LIN {X 0,Y 488.936,Z 692.562,A -85,B 0,C 180,E1 -6380.904,E2 -6380.904} C_VEL
LIN {X 0,Y 488.778,Z 691.698,A -85,B 0,C 180,E1 -6381.057,E2 -6381.057} C_VEL
LIN {X 0,Y 488.78,Z 691.596,A -85,B 0,C 180,E1 -6383.396,E2 -6383.396} C_VEL
LIN {X 0,Y 488.666,Z 691.611,A -85,B 0,C 180,E1 -6385.878,E2 -6385.878} C_VEL
LIN {X 0,Y 488.944,Z 691.579,A -85,B 0,C 180,E1 -6387.53,E2 -6387.53} C_VEL
LIN {X 0,Y 488.944,Z 691.581,A -85,B 0,C 180,E1 -6390.001,E2 -6390.001} C_VEL
LIN {X 0,Y 488.943,Z 691.584,A -85,B 0,C 180,E1 -6392.473,E2 -6392.473} C_VEL
LIN {X 0,Y 488.815,Z 691.594,A -85,B 0,C 180,E1 -6395.777,E2 -6395.777} C_VEL
LIN {X 0,Y 488.758,Z 691.602,A -85,B 0,C 180,E1 -6398.269,E2 -6398.269} C_VEL
LIN {X 0,Y 488.778,Z 691.595,A -85,B 0,C 180,E1 -6401.614,E2 -6401.614} C_VEL
LIN {X 0,Y 488.759,Z 691.601,A -85,B 0,C 180,E1 -6405.002,E2 -6405.002} C_VEL
LIN {X 0,Y 488.72,Z 691.607,A -85,B 0,C 180,E1 -6408.445,E2 -6408.445} C_VEL
LIN {X 0,Y 488.708,Z 691.61,A -85,B 0,C 180,E1 -6411.072,E2 -6411.072} C_VEL
LIN {X 0,Y 488.668,Z 691.61,A -85,B 0,C 180,E1 -6413.748,E2 -6413.748} C_VEL
LIN {X 0,Y 488.673,Z 691.604,A -85,B 0,C 180,E1 -6416.478,E2 -6416.478} C_VEL
LIN {X 0,Y 488.664,Z 691.617,A -85,B 0,C 180,E1 -6419.275,E2 -6419.275} C_VEL
LIN {X 0,Y 488.684,Z 691.605,A -85,B 0,C 180,E1 -6422.15,E2 -6422.15} C_VEL
LIN {X 0,Y 488.7,Z 691.599,A -85,B 0,C 180,E1 -6425.118,E2 -6425.118} C_VEL
LIN {X 0,Y 488.649,Z 691.611,A -85,B 0,C 180,E1 -6428.204,E2 -6428.204} C_VEL
LIN {X 0,Y 488.648,Z 691.62,A -85,B 0,C 180,E1 -6431.423,E2 -6431.423} C_VEL
LIN {X 0,Y 488.702,Z 691.606,A -85,B 0,C 180,E1 -6434.804,E2 -6434.804} C_VEL
LIN {X 0,Y 488.654,Z 691.617,A -85,B 0,C 180,E1 -6437.47,E2 -6437.47} C_VEL
LIN {X 0,Y 488.671,Z 691.61,A -85,B 0,C 180,E1 -6440.742,E2 -6440.742} C_VEL
LIN {X 0,Y 488.637,Z 691.621,A -85,B 0,C 180,E1 -6443.864,E2 -6443.864} C_VEL
LIN {X 0,Y 488.684,Z 691.61,A -85,B 0,C 180,E1 -6446.873,E2 -6446.873} C_VEL
LIN {X 0,Y 488.67,Z 691.617,A -85,B 0,C 180,E1 -6449.777,E2 -6449.777} C_VEL
LIN {X 0,Y 488.735,Z 691.812,A -85,B 0,C 180,E1 -6451.191,E2 -6451.191} C_VEL
LIN {X 0,Y 488.91,Z 692.685,A -85,B 0,C 180,E1 -6451.311,E2 -6451.311} C_VEL
LIN {X 0,Y 491.517,Z 700.39,A -85,B 0,C 180,E1 -6451.531,E2 -6451.531} C_VEL
LIN {X 0,Y 491.069,Z 767.576,A -85,B 0,C 180,E1 -6452.576,E2 -6452.576} C_VEL
LIN {X 0,Y 490.938,Z 778.889,A -85,B 0,C 180,E1 -6452.88,E2 -6452.88} C_VEL
LIN {X 0,Y 490.731,Z 789.801,A -85,B 0,C 180,E1 -6453.299,E2 -6453.299} C_VEL
LIN {X 0,Y 490.544,Z 798.848,A -85,B 0,C 180,E1 -6453.746,E2 -6453.746} C_VEL
LIN {X 0,Y 490.248,Z 807.955,A -85,B 0,C 180,E1 -6454.3,E2 -6454.3} C_VEL
LIN {X 0,Y 489.93,Z 818.39,A -85,B 0,C 180,E1 -6455.097,E2 -6455.097} C_VEL
LIN {X 0,Y 489.601,Z 826.602,A -85,B 0,C 180,E1 -6455.851,E2 -6455.851} C_VEL
LIN {X 0,Y 489.333,Z 835.233,A -85,B 0,C 180,E1 -6456.811,E2 -6456.811} C_VEL
LIN {X 0,Y 489.045,Z 842.903,A -85,B 0,C 180,E1 -6457.837,E2 -6457.837} C_VEL
LIN {X 0,Y 488.795,Z 848.474,A -85,B 0,C 180,E1 -6458.712,E2 -6458.712} C_VEL
LIN {X 0,Y 488.607,Z 854.255,A -85,B 0,C 180,E1 -6459.805,E2 -6459.805} C_VEL
LIN {X 0,Y 488.459,Z 859.764,A -85,B 0,C 180,E1 -6461.111,E2 -6461.111} C_VEL
LIN {X 0,Y 488.295,Z 864.002,A -85,B 0,C 180,E1 -6462.407,E2 -6462.407} C_VEL
LIN {X 0,Y 488.208,Z 866.278,A -85,B 0,C 180,E1 -6463.267,E2 -6463.267} C_VEL
LIN {X 0,Y 488.154,Z 868.86,A -85,B 0,C 180,E1 -6464.713,E2 -6464.713} C_VEL
LIN {X 0,Y 488.118,Z 870.091,A -85,B 0,C 180,E1 -6465.832,E2 -6465.832} C_VEL
LIN {X 0,Y 488.143,Z 870.488,A -85,B 0,C 180,E1 -6466.682,E2 -6466.682} C_VEL
LIN {X 0,Y 488.181,Z 870.191,A -85,B 0,C 180,E1 -6468.227,E2 -6468.227} C_VEL
LIN {X 0,Y 488.214,Z 869.199,A -85,B 0,C 180,E1 -6469.214,E2 -6469.214} C_VEL
LIN {X 0,Y 488.29,Z 866.395,A -85,B 0,C 180,E1 -6470.89,E2 -6470.89} C_VEL
LIN {X 0,Y 488.444,Z 863.069,A -85,B 0,C 180,E1 -6472.143,E2 -6472.143} C_VEL
LIN {X 0,Y 488.58,Z 858.666,A -85,B 0,C 180,E1 -6473.392,E2 -6473.392} C_VEL
LIN {X 0,Y 488.736,Z 853.034,A -85,B 0,C 180,E1 -6474.637,E2 -6474.637} C_VEL
LIN {X 0,Y 488.912,Z 847.33,A -85,B 0,C 180,E1 -6475.672,E2 -6475.672} C_VEL
LIN {X 0,Y 489.218,Z 840.419,A -85,B 0,C 180,E1 -6476.706,E2 -6476.706} C_VEL
LIN {X 0,Y 489.54,Z 832.033,A -85,B 0,C 180,E1 -6477.737,E2 -6477.737} C_VEL
LIN {X 0,Y 489.821,Z 824.016,A -85,B 0,C 180,E1 -6478.561,E2 -6478.561} C_VEL
LIN {X 0,Y 490.161,Z 814.265,A -85,B 0,C 180,E1 -6479.384,E2 -6479.384} C_VEL
LIN {X 0,Y 490.428,Z 805.41,A -85,B 0,C 180,E1 -6480,E2 -6480} C_VEL
LIN {X 0,Y 490.655,Z 795.361,A -85,B 0,C 180,E1 -6480.564,E2 -6480.564} C_VEL
LIN {X 0,Y 490.911,Z 784.684,A -85,B 0,C 180,E1 -6481.025,E2 -6481.025} C_VEL
LIN {X 0,Y 491.017,Z 774.27,A -85,B 0,C 180,E1 -6481.358,E2 -6481.358} C_VEL
LIN {X 0,Y 491.113,Z 762.086,A -85,B 0,C 180,E1 -6481.614,E2 -6481.614} C_VEL
LIN {X 0,Y 491.441,Z 699.545,A -85,B 0,C 180,E1 -6482.577,E2 -6482.577} C_VEL
LIN {X 0,Y 489.035,Z 692.377,A -85,B 0,C 180,E1 -6482.806,E2 -6482.806} C_VEL
LIN {X 0,Y 488.882,Z 691.641,A -85,B 0,C 180,E1 -6482.987,E2 -6482.987} C_VEL
LIN {X 0,Y 488.844,Z 691.595,A -85,B 0,C 180,E1 -6485.776,E2 -6485.776} C_VEL
LIN {X 0,Y 488.792,Z 691.601,A -85,B 0,C 180,E1 -6488.267,E2 -6488.267} C_VEL
LIN {X 0,Y 488.812,Z 691.595,A -85,B 0,C 180,E1 -6491.612,E2 -6491.612} C_VEL
LIN {X 0,Y 488.769,Z 691.6,A -85,B 0,C 180,E1 -6495,E2 -6495} C_VEL
LIN {X 0,Y 488.754,Z 691.607,A -85,B 0,C 180,E1 -6498.442,E2 -6498.442} C_VEL
LIN {X 0,Y 488.714,Z 691.607,A -85,B 0,C 180,E1 -6501.07,E2 -6501.07} C_VEL
LIN {X 0,Y 488.69,Z 691.607,A -85,B 0,C 180,E1 -6503.746,E2 -6503.746} C_VEL
LIN {X 0,Y 488.732,Z 691.609,A -85,B 0,C 180,E1 -6506.928,E2 -6506.928} C_VEL
LIN {X 0,Y 488.731,Z 691.604,A -85,B 0,C 180,E1 -6510.219,E2 -6510.219} C_VEL
LIN {X 0,Y 488.735,Z 691.604,A -85,B 0,C 180,E1 -6513.483,E2 -6513.483} C_VEL
LIN {X 0,Y 488.688,Z 691.609,A -85,B 0,C 180,E1 -6516.354,E2 -6516.354} C_VEL
LIN {X 0,Y 488.707,Z 691.612,A -85,B 0,C 180,E1 -6519.254,E2 -6519.254} C_VEL
LIN {X 0,Y 488.713,Z 691.609,A -85,B 0,C 180,E1 -6521.599,E2 -6521.599} C_VEL
LIN {X 0,Y 488.708,Z 691.608,A -85,B 0,C 180,E1 -6524.802,E2 -6524.802} C_VEL
LIN {X 0,Y 488.698,Z 691.614,A -85,B 0,C 180,E1 -6527.474,E2 -6527.474} C_VEL
LIN {X 0,Y 488.739,Z 691.607,A -85,B 0,C 180,E1 -6529.676,E2 -6529.676} C_VEL
LIN {X 0,Y 488.676,Z 691.61,A -85,B 0,C 180,E1 -6532.84,E2 -6532.84} C_VEL
LIN {X 0,Y 488.729,Z 691.609,A -85,B 0,C 180,E1 -6535.886,E2 -6535.886} C_VEL
LIN {X 0,Y 488.698,Z 691.612,A -85,B 0,C 180,E1 -6538.819,E2 -6538.819} C_VEL
LIN {X 0,Y 488.803,Z 691.843,A -85,B 0,C 180,E1 -6540.068,E2 -6540.068} C_VEL
LIN {X 0,Y 492.608,Z 708.802,A -85,B 0,C 180,E1 -6542.527,E2 -6542.527} C_VEL
LIN {X 0,Y 491.674,Z 731.997,A -85,B 0,C 180,E1 -6545.509,E2 -6545.509} C_VEL
LIN {X 0,Y 490.938,Z 754.807,A -85,B 0,C 180,E1 -6548.401,E2 -6548.401} C_VEL
LIN {X 0,Y 490.099,Z 782.413,A -85,B 0,C 180,E1 -6551.825,E2 -6551.825} C_VEL
LIN {X 0,Y 489.619,Z 797.491,A -85,B 0,C 180,E1 -6553.682,E2 -6553.682} C_VEL
LIN {X 0,Y 490.629,Z 806.708,A -85,B 0,C 180,E1 -6553.883,E2 -6553.883} C_VEL
LIN {X 0,Y 491.648,Z 815.903,A -85,B 0,C 180,E1 -6554.053,E2 -6554.053} C_VEL
LIN {X 0,Y 491.061,Z 909.011,A -85,B 0,C 180,E1 -6555.441,E2 -6555.441} C_VEL
LIN {X 0,Y 490.661,Z 922.838,A -85,B 0,C 180,E1 -6555.826,E2 -6555.826} C_VEL
LIN {X 0,Y 490.322,Z 935.816,A -85,B 0,C 180,E1 -6556.372,E2 -6556.372} C_VEL
LIN {X 0,Y 489.911,Z 948.159,A -85,B 0,C 180,E1 -6557.077,E2 -6557.077} C_VEL
LIN {X 0,Y 489.566,Z 959.167,A -85,B 0,C 180,E1 -6557.879,E2 -6557.879} C_VEL
LIN {X 0,Y 489.119,Z 969.532,A -85,B 0,C 180,E1 -6558.814,E2 -6558.814} C_VEL
LIN {X 0,Y 488.807,Z 978.886,A -85,B 0,C 180,E1 -6559.854,E2 -6559.854} C_VEL
LIN {X 0,Y 488.488,Z 988.009,A -85,B 0,C 180,E1 -6561.102,E2 -6561.102} C_VEL
LIN {X 0,Y 488.265,Z 995.37,A -85,B 0,C 180,E1 -6562.348,E2 -6562.348} C_VEL
LIN {X 0,Y 488.141,Z 1001.708,A -85,B 0,C 180,E1 -6563.703,E2 -6563.703} C_VEL
LIN {X 0,Y 488.037,Z 1006.546,A -85,B 0,C 180,E1 -6565.042,E2 -6565.042} C_VEL
LIN {X 0,Y 488.031,Z 1008.908,A -85,B 0,C 180,E1 -6565.87,E2 -6565.87} C_VEL
LIN {X 0,Y 488.029,Z 1010.823,A -85,B 0,C 180,E1 -6566.697,E2 -6566.697} C_VEL
LIN {X 0,Y 487.977,Z 1012.255,A -85,B 0,C 180,E1 -6567.522,E2 -6567.522} C_VEL
LIN {X 0,Y 487.951,Z 1013.276,A -85,B 0,C 180,E1 -6568.348,E2 -6568.348} C_VEL
LIN {X 0,Y 487.913,Z 1013.895,A -85,B 0,C 180,E1 -6569.173,E2 -6569.173} C_VEL
LIN {X 0,Y 487.905,Z 1014.113,A -85,B 0,C 180,E1 -6569.999,E2 -6569.999} C_VEL
LIN {X 0,Y 487.914,Z 1013.89,A -85,B 0,C 180,E1 -6570.824,E2 -6570.824} C_VEL
LIN {X 0,Y 487.952,Z 1013.268,A -85,B 0,C 180,E1 -6571.649,E2 -6571.649} C_VEL
LIN {X 0,Y 487.978,Z 1012.243,A -85,B 0,C 180,E1 -6572.475,E2 -6572.475} C_VEL
LIN {X 0,Y 488.028,Z 1010.805,A -85,B 0,C 180,E1 -6573.301,E2 -6573.301} C_VEL
LIN {X 0,Y 488.02,Z 1007.773,A -85,B 0,C 180,E1 -6574.542,E2 -6574.542} C_VEL
LIN {X 0,Y 488.139,Z 1003.69,A -85,B 0,C 180,E1 -6575.783,E2 -6575.783} C_VEL
LIN {X 0,Y 488.188,Z 997.396,A -85,B 0,C 180,E1 -6577.235,E2 -6577.235} C_VEL
LIN {X 0,Y 488.418,Z 990.553,A -85,B 0,C 180,E1 -6578.48,E2 -6578.48} C_VEL
LIN {X 0,Y 488.674,Z 982.07,A -85,B 0,C 180,E1 -6579.728,E2 -6579.728} C_VEL
LIN {X 0,Y 488.946,Z 973.387,A -85,B 0,C 180,E1 -6580.768,E2 -6580.768} C_VEL
LIN {X 0,Y 489.38,Z 962.702,A -85,B 0,C 180,E1 -6581.807,E2 -6581.807} C_VEL
LIN {X 0,Y 489.823,Z 951.136,A -85,B 0,C 180,E1 -6582.711,E2 -6582.711} C_VEL
LIN {X 0,Y 490.176,Z 938.635,A -85,B 0,C 180,E1 -6583.472,E2 -6583.472} C_VEL
LIN {X 0,Y 490.612,Z 926.141,A -85,B 0,C 180,E1 -6584.04,E2 -6584.04} C_VEL
LIN {X 0,Y 490.952,Z 913.323,A -85,B 0,C 180,E1 -6584.454,E2 -6584.454} C_VEL
LIN {X 0,Y 491.139,Z 898.092,A -85,B 0,C 180,E1 -6584.739,E2 -6584.739} C_VEL
LIN {X 0,Y 491.615,Z 814.3,A -85,B 0,C 180,E1 -6585.966,E2 -6585.966} C_VEL
LIN {X 0,Y 489.61,Z 797.388,A -85,B 0,C 180,E1 -6586.296,E2 -6586.296} C_VEL
LIN {X 0,Y 490.203,Z 775.247,A -85,B 0,C 180,E1 -6588.998,E2 -6588.998} C_VEL
LIN {X 0,Y 490.964,Z 750.475,A -85,B 0,C 180,E1 -6592.07,E2 -6592.07} C_VEL
LIN {X 0,Y 491.789,Z 726.02,A -85,B 0,C 180,E1 -6595.158,E2 -6595.158} C_VEL
LIN {X 0,Y 492.452,Z 708.982,A -85,B 0,C 180,E1 -6597.346,E2 -6597.346} C_VEL
LIN {X 0,Y 490.614,Z 699.96,A -85,B 0,C 180,E1 -6598.62,E2 -6598.62} C_VEL
LIN {X 0,Y 488.756,Z 691.718,A -85,B 0,C 180,E1 -6599.859,E2 -6599.859} C_VEL
LIN {X 0,Y 488.733,Z 691.605,A -85,B 0,C 180,E1 -6603.121,E2 -6603.121} C_VEL
LIN {X 0,Y 488.671,Z 691.616,A -85,B 0,C 180,E1 -6606.131,E2 -6606.131} C_VEL
LIN {X 0,Y 488.694,Z 691.609,A -85,B 0,C 180,E1 -6609.253,E2 -6609.253} C_VEL
LIN {X 0,Y 488.699,Z 691.607,A -85,B 0,C 180,E1 -6611.599,E2 -6611.599} C_VEL
LIN {X 0,Y 488.704,Z 691.612,A -85,B 0,C 180,E1 -6614.8,E2 -6614.8} C_VEL
LIN {X 0,Y 488.688,Z 691.609,A -85,B 0,C 180,E1 -6617.474,E2 -6617.474} C_VEL
LIN {X 0,Y 488.724,Z 691.598,A -85,B 0,C 180,E1 -6619.676,E2 -6619.676} C_VEL
LIN {X 0,Y 488.673,Z 691.616,A -85,B 0,C 180,E1 -6622.84,E2 -6622.84} C_VEL
LIN {X 0,Y 488.725,Z 691.602,A -85,B 0,C 180,E1 -6625.887,E2 -6625.887} C_VEL
LIN {X 0,Y 488.685,Z 691.61,A -85,B 0,C 180,E1 -6628.82,E2 -6628.82} C_VEL
LIN {X 0,Y 488.736,Z 691.604,A -85,B 0,C 180,E1 -6631.671,E2 -6631.671} C_VEL
LIN {X 0,Y 488.74,Z 691.6,A -85,B 0,C 180,E1 -6634.444,E2 -6634.444} C_VEL
LIN {X 0,Y 488.71,Z 691.608,A -85,B 0,C 180,E1 -6637.153,E2 -6637.153} C_VEL
LIN {X 0,Y 488.713,Z 691.611,A -85,B 0,C 180,E1 -6639.81,E2 -6639.81} C_VEL
LIN {X 0,Y 488.722,Z 691.6,A -85,B 0,C 180,E1 -6642.423,E2 -6642.423} C_VEL
LIN {X 0,Y 488.75,Z 691.6,A -85,B 0,C 180,E1 -6644.999,E2 -6644.999} C_VEL
LIN {X 0,Y 488.793,Z 691.597,A -85,B 0,C 180,E1 -6648.387,E2 -6648.387} C_VEL
LIN {X 0,Y 488.805,Z 691.592,A -85,B 0,C 180,E1 -6651.734,E2 -6651.734} C_VEL
LIN {X 0,Y 488.836,Z 691.594,A -85,B 0,C 180,E1 -6654.224,E2 -6654.224} C_VEL
LIN {X 0,Y 488.948,Z 691.574,A -85,B 0,C 180,E1 -6657.529,E2 -6657.529} C_VEL
LIN {X 0,Y 488.943,Z 691.577,A -85,B 0,C 180,E1 -6660.824,E2 -6660.824} C_VEL
LIN {X 0,Y 488.948,Z 691.583,A -85,B 0,C 180,E1 -6662.472,E2 -6662.472} C_VEL
LIN {X 0,Y 488.836,Z 691.588,A -85,B 0,C 180,E1 -6665.776,E2 -6665.776} C_VEL
LIN {X 0,Y 488.806,Z 691.595,A -85,B 0,C 180,E1 -6668.267,E2 -6668.267} C_VEL
LIN {X 0,Y 488.796,Z 691.593,A -85,B 0,C 180,E1 -6671.613,E2 -6671.613} C_VEL
LIN {X 0,Y 488.75,Z 691.605,A -85,B 0,C 180,E1 -6675.001,E2 -6675.001} C_VEL
LIN {X 0,Y 488.735,Z 691.603,A -85,B 0,C 180,E1 -6678.443,E2 -6678.443} C_VEL
LIN {X 0,Y 488.695,Z 691.615,A -85,B 0,C 180,E1 -6681.072,E2 -6681.072} C_VEL
LIN {X 0,Y 488.661,Z 691.608,A -85,B 0,C 180,E1 -6683.747,E2 -6683.747} C_VEL
LIN {X 0,Y 488.737,Z 691.606,A -85,B 0,C 180,E1 -6686.934,E2 -6686.934} C_VEL
LIN {X 0,Y 488.712,Z 691.605,A -85,B 0,C 180,E1 -6689.271,E2 -6689.271} C_VEL
LIN {X 0,Y 488.694,Z 691.604,A -85,B 0,C 180,E1 -6692.148,E2 -6692.148} C_VEL
LIN {X 0,Y 488.713,Z 691.608,A -85,B 0,C 180,E1 -6695.116,E2 -6695.116} C_VEL
LIN {X 0,Y 488.672,Z 691.61,A -85,B 0,C 180,E1 -6698.201,E2 -6698.201} C_VEL
LIN {X 0,Y 488.71,Z 691.607,A -85,B 0,C 180,E1 -6700.346,E2 -6700.346} C_VEL
LIN {X 0,Y 488.677,Z 691.614,A -85,B 0,C 180,E1 -6703.656,E2 -6703.656} C_VEL
LIN {X 0,Y 488.671,Z 691.609,A -85,B 0,C 180,E1 -6706.346,E2 -6706.346} C_VEL
LIN {X 0,Y 488.772,Z 691.798,A -85,B 0,C 180,E1 -6709.048,E2 -6709.048} C_VEL
LIN {X 0,Y 489.014,Z 692.905,A -85,B 0,C 180,E1 -6709.184,E2 -6709.184} C_VEL
LIN {X 0,Y 491.909,Z 700.992,A -85,B 0,C 180,E1 -6709.415,E2 -6709.415} C_VEL
LIN {X 0,Y 491.437,Z 772.238,A -85,B 0,C 180,E1 -6710.494,E2 -6710.494} C_VEL
LIN {X 0,Y 491.368,Z 785.777,A -85,B 0,C 180,E1 -6710.878,E2 -6710.878} C_VEL
LIN {X 0,Y 491.208,Z 797.787,A -85,B 0,C 180,E1 -6711.381,E2 -6711.381} C_VEL
LIN {X 0,Y 490.972,Z 807.684,A -85,B 0,C 180,E1 -6711.928,E2 -6711.928} C_VEL
LIN {X 0,Y 490.236,Z 812.918,A -85,B 0,C 180,E1 -6712.238,E2 -6712.238} C_VEL
LIN {X 0,Y 487.217,Z 821.277,A -85,B 0,C 180,E1 -6712.758,E2 -6712.758} C_VEL
LIN {X 0,Y 484.13,Z 829.158,A -85,B 0,C 180,E1 -6713.365,E2 -6713.365} C_VEL
LIN {X 0,Y 483.294,Z 833.637,A -85,B 0,C 180,E1 -6713.808,E2 -6713.808} C_VEL
LIN {X 0,Y 482.865,Z 842.864,A -85,B 0,C 180,E1 -6714.908,E2 -6714.908} C_VEL
LIN {X 0,Y 482.444,Z 851.205,A -85,B 0,C 180,E1 -6716.135,E2 -6716.135} C_VEL
LIN {X 0,Y 482.214,Z 857.921,A -85,B 0,C 180,E1 -6717.369,E2 -6717.369} C_VEL
LIN {X 0,Y 481.878,Z 864.127,A -85,B 0,C 180,E1 -6718.82,E2 -6718.82} C_VEL
LIN {X 0,Y 481.67,Z 868.785,A -85,B 0,C 180,E1 -6720.26,E2 -6720.26} C_VEL
LIN {X 0,Y 481.557,Z 871.112,A -85,B 0,C 180,E1 -6721.211,E2 -6721.211} C_VEL
LIN {X 0,Y 481.484,Z 872.871,A -85,B 0,C 180,E1 -6722.156,E2 -6722.156} C_VEL
LIN {X 0,Y 481.455,Z 874.126,A -85,B 0,C 180,E1 -6723.096,E2 -6723.096} C_VEL
LIN {X 0,Y 481.39,Z 874.851,A -85,B 0,C 180,E1 -6724.026,E2 -6724.026} C_VEL
LIN {X 0,Y 481.378,Z 875.127,A -85,B 0,C 180,E1 -6724.953,E2 -6724.953} C_VEL
LIN {X 0,Y 481.359,Z 874.918,A -85,B 0,C 180,E1 -6725.872,E2 -6725.872} C_VEL
LIN {X 0,Y 481.396,Z 874.137,A -85,B 0,C 180,E1 -6726.891,E2 -6726.891} C_VEL
LIN {X 0,Y 481.44,Z 873.13,A -85,B 0,C 180,E1 -6727.696,E2 -6727.696} C_VEL
LIN {X 0,Y 481.603,Z 870.535,A -85,B 0,C 180,E1 -6729.06,E2 -6729.06} C_VEL
LIN {X 0,Y 481.73,Z 866.893,A -85,B 0,C 180,E1 -6730.396,E2 -6730.396} C_VEL
LIN {X 0,Y 481.967,Z 861.718,A -85,B 0,C 180,E1 -6731.804,E2 -6731.804} C_VEL
LIN {X 0,Y 482.226,Z 854.725,A -85,B 0,C 180,E1 -6733.273,E2 -6733.273} C_VEL
LIN {X 0,Y 482.587,Z 847.687,A -85,B 0,C 180,E1 -6734.441,E2 -6734.441} C_VEL
LIN {X 0,Y 482.958,Z 838.437,A -85,B 0,C 180,E1 -6735.679,E2 -6735.679} C_VEL
LIN {X 0,Y 483.355,Z 829.161,A -85,B 0,C 180,E1 -6736.684,E2 -6736.684} C_VEL
LIN {X 0,Y 483.733,Z 818.409,A -85,B 0,C 180,E1 -6737.627,E2 -6737.627} C_VEL
LIN {X 0,Y 484.076,Z 807.541,A -85,B 0,C 180,E1 -6738.38,E2 -6738.38} C_VEL
LIN {X 0,Y 484.32,Z 795.637,A -85,B 0,C 180,E1 -6739.022,E2 -6739.022} C_VEL
LIN {X 0,Y 484.505,Z 782.745,A -85,B 0,C 180,E1 -6739.528,E2 -6739.528} C_VEL
LIN {X 0,Y 484.6,Z 770.059,A -85,B 0,C 180,E1 -6739.847,E2 -6739.847} C_VEL
LIN {X 0,Y 484.959,Z 702.07,A -85,B 0,C 180,E1 -6740.876,E2 -6740.876} C_VEL
LIN {X 0,Y 481.891,Z 693.353,A -85,B 0,C 180,E1 -6741.148,E2 -6741.148} C_VEL
LIN {X 0,Y 481.733,Z 692.534,A -85,B 0,C 180,E1 -6741.327,E2 -6741.327} C_VEL
LIN {X 0,Y 481.777,Z 692.474,A -85,B 0,C 180,E1 -6744.14,E2 -6744.14} C_VEL
LIN {X 0,Y 481.909,Z 692.456,A -85,B 0,C 180,E1 -6747.494,E2 -6747.494} C_VEL
LIN {X 0,Y 481.913,Z 692.457,A -85,B 0,C 180,E1 -6750.001,E2 -6750.001} C_VEL
LIN {X 0,Y 481.908,Z 692.46,A -85,B 0,C 180,E1 -6752.509,E2 -6752.509} C_VEL
LIN {X 0,Y 481.777,Z 692.471,A -85,B 0,C 180,E1 -6755.862,E2 -6755.862} C_VEL
LIN {X 0,Y 481.716,Z 692.481,A -85,B 0,C 180,E1 -6758.39,E2 -6758.39} C_VEL
LIN {X 0,Y 481.729,Z 692.473,A -85,B 0,C 180,E1 -6761.787,E2 -6761.787} C_VEL
LIN {X 0,Y 481.743,Z 692.472,A -85,B 0,C 180,E1 -6765.225,E2 -6765.225} C_VEL
LIN {X 0,Y 481.663,Z 692.487,A -85,B 0,C 180,E1 -6768.725,E2 -6768.725} C_VEL
LIN {X 0,Y 481.647,Z 692.486,A -85,B 0,C 180,E1 -6771.396,E2 -6771.396} C_VEL
LIN {X 0,Y 481.647,Z 692.484,A -85,B 0,C 180,E1 -6774.116,E2 -6774.116} C_VEL
LIN {X 0,Y 481.647,Z 692.483,A -85,B 0,C 180,E1 -6777.115,E2 -6777.115} C_VEL
LIN {X 0,Y 481.605,Z 692.491,A -85,B 0,C 180,E1 -6779.747,E2 -6779.747} C_VEL
LIN {X 0,Y 481.639,Z 692.484,A -85,B 0,C 180,E1 -6782.678,E2 -6782.678} C_VEL
LIN {X 0,Y 481.644,Z 692.478,A -85,B 0,C 180,E1 -6785.2,E2 -6785.2} C_VEL
LIN {X 0,Y 481.626,Z 692.487,A -85,B 0,C 180,E1 -6788.002,E2 -6788.002} C_VEL
LIN {X 0,Y 481.609,Z 692.491,A -85,B 0,C 180,E1 -6791.048,E2 -6791.048} C_VEL
LIN {X 0,Y 481.638,Z 692.485,A -85,B 0,C 180,E1 -6794.461,E2 -6794.461} C_VEL
LIN {X 0,Y 481.618,Z 692.488,A -85,B 0,C 180,E1 -6796.856,E2 -6796.856} C_VEL
LIN {X 0,Y 481.633,Z 692.492,A -85,B 0,C 180,E1 -6800.055,E2 -6800.055} C_VEL
LIN {X 0,Y 481.602,Z 692.492,A -85,B 0,C 180,E1 -6803.251,E2 -6803.251} C_VEL
LIN {X 0,Y 481.678,Z 692.487,A -85,B 0,C 180,E1 -6806.327,E2 -6806.327} C_VEL
LIN {X 0,Y 481.617,Z 692.494,A -85,B 0,C 180,E1 -6809.426,E2 -6809.426} C_VEL
LIN {X 0,Y 481.68,Z 692.657,A -85,B 0,C 180,E1 -6810.951,E2 -6810.951} C_VEL
LIN {X 0,Y 481.895,Z 693.673,A -85,B 0,C 180,E1 -6811.09,E2 -6811.09} C_VEL
LIN {X 0,Y 484.721,Z 701.805,A -85,B 0,C 180,E1 -6811.327,E2 -6811.327} C_VEL
LIN {X 0,Y 484.189,Z 768.388,A -85,B 0,C 180,E1 -6812.382,E2 -6812.382} C_VEL
LIN {X 0,Y 484.073,Z 779.919,A -85,B 0,C 180,E1 -6812.697,E2 -6812.697} C_VEL
LIN {X 0,Y 483.85,Z 790.799,A -85,B 0,C 180,E1 -6813.121,E2 -6813.121} C_VEL
LIN {X 0,Y 483.662,Z 799.838,A -85,B 0,C 180,E1 -6813.576,E2 -6813.576} C_VEL
LIN {X 0,Y 483.368,Z 808.945,A -85,B 0,C 180,E1 -6814.139,E2 -6814.139} C_VEL
LIN {X 0,Y 483.062,Z 818.474,A -85,B 0,C 180,E1 -6814.866,E2 -6814.866} C_VEL
LIN {X 0,Y 482.688,Z 827.593,A -85,B 0,C 180,E1 -6815.712,E2 -6815.712} C_VEL
LIN {X 0,Y 482.43,Z 835.608,A -85,B 0,C 180,E1 -6816.605,E2 -6816.605} C_VEL
LIN {X 0,Y 482.175,Z 842.456,A -85,B 0,C 180,E1 -6817.504,E2 -6817.504} C_VEL
LIN {X 0,Y 481.819,Z 849.481,A -85,B 0,C 180,E1 -6818.613,E2 -6818.613} C_VEL
LIN {X 0,Y 481.657,Z 854.26,A -85,B 0,C 180,E1 -6819.501,E2 -6819.501} C_VEL
LIN {X 0,Y 481.498,Z 860.012,A -85,B 0,C 180,E1 -6820.827,E2 -6820.827} C_VEL
LIN {X 0,Y 481.32,Z 864.44,A -85,B 0,C 180,E1 -6822.143,E2 -6822.143} C_VEL
LIN {X 0,Y 481.205,Z 866.797,A -85,B 0,C 180,E1 -6823.016,E2 -6823.016} C_VEL
LIN {X 0,Y 481.141,Z 869.948,A -85,B 0,C 180,E1 -6824.756,E2 -6824.756} C_VEL
LIN {X 0,Y 481.1,Z 870.954,A -85,B 0,C 180,E1 -6825.621,E2 -6825.621} C_VEL
LIN {X 0,Y 481.122,Z 871.467,A -85,B 0,C 180,E1 -6826.484,E2 -6826.484} C_VEL
LIN {X 0,Y 481.179,Z 871.245,A -85,B 0,C 180,E1 -6828.201,E2 -6828.201} C_VEL
LIN {X 0,Y 481.224,Z 869.341,A -85,B 0,C 180,E1 -6829.906,E2 -6829.906} C_VEL
LIN {X 0,Y 481.301,Z 866.839,A -85,B 0,C 180,E1 -6831.18,E2 -6831.18} C_VEL
LIN {X 0,Y 481.489,Z 863.306,A -85,B 0,C 180,E1 -6832.451,E2 -6832.451} C_VEL
LIN {X 0,Y 481.652,Z 858.673,A -85,B 0,C 180,E1 -6833.717,E2 -6833.717} C_VEL
LIN {X 0,Y 481.779,Z 853.92,A -85,B 0,C 180,E1 -6834.769,E2 -6834.769} C_VEL
LIN {X 0,Y 481.98,Z 848.169,A -85,B 0,C 180,E1 -6835.819,E2 -6835.819} C_VEL
LIN {X 0,Y 482.311,Z 841.203,A -85,B 0,C 180,E1 -6836.867,E2 -6836.867} C_VEL
LIN {X 0,Y 482.642,Z 832.757,A -85,B 0,C 180,E1 -6837.914,E2 -6837.914} C_VEL
LIN {X 0,Y 482.951,Z 824.664,A -85,B 0,C 180,E1 -6838.749,E2 -6838.749} C_VEL
LIN {X 0,Y 483.236,Z 816.234,A -85,B 0,C 180,E1 -6839.479,E2 -6839.479} C_VEL
LIN {X 0,Y 483.532,Z 807.575,A -85,B 0,C 180,E1 -6840.104,E2 -6840.104} C_VEL
LIN {X 0,Y 483.785,Z 796.73,A -85,B 0,C 180,E1 -6840.728,E2 -6840.728} C_VEL
LIN {X 0,Y 484.018,Z 786.174,A -85,B 0,C 180,E1 -6841.196,E2 -6841.196} C_VEL
LIN {X 0,Y 484.139,Z 775.934,A -85,B 0,C 180,E1 -6841.534,E2 -6841.534} C_VEL
LIN {X 0,Y 484.266,Z 762.405,A -85,B 0,C 180,E1 -6841.819,E2 -6841.819} C_VEL
LIN {X 0,Y 484.709,Z 701.263,A -85,B 0,C 180,E1 -6842.78,E2 -6842.78} C_VEL
LIN {X 0,Y 482.024,Z 693.475,A -85,B 0,C 180,E1 -6843.02,E2 -6843.02} C_VEL
LIN {X 0,Y 481.805,Z 692.564,A -85,B 0,C 180,E1 -6843.183,E2 -6843.183} C_VEL
LIN {X 0,Y 481.803,Z 692.473,A -85,B 0,C 180,E1 -6845.86,E2 -6845.86} C_VEL
LIN {X 0,Y 481.746,Z 692.478,A -85,B 0,C 180,E1 -6848.388,E2 -6848.388} C_VEL
LIN {X 0,Y 481.758,Z 692.475,A -85,B 0,C 180,E1 -6851.785,E2 -6851.785} C_VEL
LIN {X 0,Y 481.75,Z 692.473,A -85,B 0,C 180,E1 -6855.224,E2 -6855.224} C_VEL
LIN {X 0,Y 481.715,Z 692.482,A -85,B 0,C 180,E1 -6858.722,E2 -6858.722} C_VEL
LIN {X 0,Y 481.652,Z 692.485,A -85,B 0,C 180,E1 -6861.394,E2 -6861.394} C_VEL
LIN {X 0,Y 481.67,Z 692.484,A -85,B 0,C 180,E1 -6864.113,E2 -6864.113} C_VEL
LIN {X 0,Y 481.701,Z 692.482,A -85,B 0,C 180,E1 -6867.126,E2 -6867.126} C_VEL
LIN {X 0,Y 481.68,Z 692.481,A -85,B 0,C 180,E1 -6869.741,E2 -6869.741} C_VEL
LIN {X 0,Y 481.677,Z 692.486,A -85,B 0,C 180,E1 -6872.674,E2 -6872.674} C_VEL
LIN {X 0,Y 481.642,Z 692.487,A -85,B 0,C 180,E1 -6875.709,E2 -6875.709} C_VEL
LIN {X 0,Y 481.677,Z 692.487,A -85,B 0,C 180,E1 -6878.859,E2 -6878.859} C_VEL
LIN {X 0,Y 481.659,Z 692.485,A -85,B 0,C 180,E1 -6881.912,E2 -6881.912} C_VEL
LIN {X 0,Y 481.661,Z 692.484,A -85,B 0,C 180,E1 -6884.457,E2 -6884.457} C_VEL
LIN {X 0,Y 481.654,Z 692.487,A -85,B 0,C 180,E1 -6887.839,E2 -6887.839} C_VEL
LIN {X 0,Y 481.663,Z 692.483,A -85,B 0,C 180,E1 -6890.654,E2 -6890.654} C_VEL
LIN {X 0,Y 481.628,Z 692.493,A -85,B 0,C 180,E1 -6893.376,E2 -6893.376} C_VEL
LIN {X 0,Y 481.682,Z 692.485,A -85,B 0,C 180,E1 -6896.327,E2 -6896.327} C_VEL
LIN {X 0,Y 481.731,Z 692.662,A -85,B 0,C 180,E1 -6899.809,E2 -6899.809} C_VEL
LIN {X 0,Y 485.708,Z 710.28,A -85,B 0,C 180,E1 -6902.416,E2 -6902.416} C_VEL
LIN {X 0,Y 484.681,Z 734.593,A -85,B 0,C 180,E1 -6905.589,E2 -6905.589} C_VEL
LIN {X 0,Y 483.88,Z 757.058,A -85,B 0,C 180,E1 -6908.475,E2 -6908.475} C_VEL
LIN {X 0,Y 482.979,Z 784.87,A -85,B 0,C 180,E1 -6911.987,E2 -6911.987} C_VEL
LIN {X 0,Y 482.603,Z 796.784,A -85,B 0,C 180,E1 -6913.458,E2 -6913.458} C_VEL
LIN {X 0,Y 484.798,Z 816.369,A -85,B 0,C 180,E1 -6913.843,E2 -6913.843} C_VEL
LIN {X 0,Y 484.168,Z 907.958,A -85,B 0,C 180,E1 -6915.229,E2 -6915.229} C_VEL
LIN {X 0,Y 483.763,Z 921.804,A -85,B 0,C 180,E1 -6915.62,E2 -6915.62} C_VEL
LIN {X 0,Y 483.37,Z 934.791,A -85,B 0,C 180,E1 -6916.172,E2 -6916.172} C_VEL
LIN {X 0,Y 482.917,Z 947.141,A -85,B 0,C 180,E1 -6916.887,E2 -6916.887} C_VEL
LIN {X 0,Y 482.538,Z 958.144,A -85,B 0,C 180,E1 -6917.7,E2 -6917.7} C_VEL
LIN {X 0,Y 482.112,Z 968.519,A -85,B 0,C 180,E1 -6918.649,E2 -6918.649} C_VEL
LIN {X 0,Y 481.728,Z 977.867,A -85,B 0,C 180,E1 -6919.704,E2 -6919.704} C_VEL
LIN {X 0,Y 481.423,Z 986.996,A -85,B 0,C 180,E1 -6920.97,E2 -6920.97} C_VEL
LIN {X 0,Y 481.209,Z 994.362,A -85,B 0,C 180,E1 -6922.235,E2 -6922.235} C_VEL
LIN {X 0,Y 481.077,Z 1001.041,A -85,B 0,C 180,E1 -6923.696,E2 -6923.696} C_VEL
LIN {X 0,Y 480.999,Z 1005.544,A -85,B 0,C 180,E1 -6924.969,E2 -6924.969} C_VEL
LIN {X 0,Y 480.976,Z 1007.903,A -85,B 0,C 180,E1 -6925.809,E2 -6925.809} C_VEL
LIN {X 0,Y 480.984,Z 1009.82,A -85,B 0,C 180,E1 -6926.648,E2 -6926.648} C_VEL
LIN {X 0,Y 480.938,Z 1011.252,A -85,B 0,C 180,E1 -6927.486,E2 -6927.486} C_VEL
LIN {X 0,Y 480.916,Z 1012.273,A -85,B 0,C 180,E1 -6928.324,E2 -6928.324} C_VEL
LIN {X 0,Y 480.883,Z 1012.89,A -85,B 0,C 180,E1 -6929.161,E2 -6929.161} C_VEL
LIN {X 0,Y 480.878,Z 1013.107,A -85,B 0,C 180,E1 -6929.999,E2 -6929.999} C_VEL
LIN {X 0,Y 480.885,Z 1012.882,A -85,B 0,C 180,E1 -6930.836,E2 -6930.836} C_VEL
LIN {X 0,Y 480.919,Z 1012.257,A -85,B 0,C 180,E1 -6931.674,E2 -6931.674} C_VEL
LIN {X 0,Y 480.941,Z 1011.227,A -85,B 0,C 180,E1 -6932.511,E2 -6932.511} C_VEL
LIN {X 0,Y 480.983,Z 1009.786,A -85,B 0,C 180,E1 -6933.349,E2 -6933.349} C_VEL
LIN {X 0,Y 480.975,Z 1006.748,A -85,B 0,C 180,E1 -6934.608,E2 -6934.608} C_VEL
LIN {X 0,Y 481.078,Z 1002.657,A -85,B 0,C 180,E1 -6935.868,E2 -6935.868} C_VEL
LIN {X 0,Y 481.151,Z 996.358,A -85,B 0,C 180,E1 -6937.342,E2 -6937.342} C_VEL
LIN {X 0,Y 481.356,Z 989.503,A -85,B 0,C 180,E1 -6938.606,E2 -6938.606} C_VEL
LIN {X 0,Y 481.607,Z 981.009,A -85,B 0,C 180,E1 -6939.872,E2 -6939.872} C_VEL
LIN {X 0,Y 481.931,Z 972.324,A -85,B 0,C 180,E1 -6940.927,E2 -6940.927} C_VEL
LIN {X 0,Y 482.387,Z 961.632,A -85,B 0,C 180,E1 -6941.981,E2 -6941.981} C_VEL
LIN {X 0,Y 482.838,Z 949.769,A -85,B 0,C 180,E1 -6942.919,E2 -6942.919} C_VEL
LIN {X 0,Y 483.205,Z 937.542,A -85,B 0,C 180,E1 -6943.67,E2 -6943.67} C_VEL
LIN {X 0,Y 483.683,Z 925.039,A -85,B 0,C 180,E1 -6944.246,E2 -6944.246} C_VEL
LIN {X 0,Y 484.031,Z 912.198,A -85,B 0,C 180,E1 -6944.665,E2 -6944.665} C_VEL
LIN {X 0,Y 484.259,Z 898.711,A -85,B 0,C 180,E1 -6944.927,E2 -6944.927} C_VEL
LIN {X 0,Y 484.665,Z 814.217,A -85,B 0,C 180,E1 -6946.186,E2 -6946.186} C_VEL
LIN {X 0,Y 482.581,Z 796.299,A -85,B 0,C 180,E1 -6946.54,E2 -6946.54} C_VEL
LIN {X 0,Y 483.176,Z 774.701,A -85,B 0,C 180,E1 -6949.215,E2 -6949.215} C_VEL
LIN {X 0,Y 483.972,Z 751.215,A -85,B 0,C 180,E1 -6952.181,E2 -6952.181} C_VEL
LIN {X 0,Y 484.869,Z 726.818,A -85,B 0,C 180,E1 -6955.313,E2 -6955.313} C_VEL
LIN {X 0,Y 485.494,Z 709.373,A -85,B 0,C 180,E1 -6957.594,E2 -6957.594} C_VEL
LIN {X 0,Y 481.719,Z 692.624,A -85,B 0,C 180,E1 -6960.083,E2 -6960.083} C_VEL
LIN {X 0,Y 481.692,Z 692.479,A -85,B 0,C 180,E1 -6963.732,E2 -6963.732} C_VEL
LIN {X 0,Y 481.619,Z 692.495,A -85,B 0,C 180,E1 -6966.746,E2 -6966.746} C_VEL
LIN {X 0,Y 481.67,Z 692.484,A -85,B 0,C 180,E1 -6969.939,E2 -6969.939} C_VEL
LIN {X 0,Y 481.631,Z 692.487,A -85,B 0,C 180,E1 -6973.299,E2 -6973.299} C_VEL
LIN {X 0,Y 481.673,Z 692.484,A -85,B 0,C 180,E1 -6976.704,E2 -6976.704} C_VEL
LIN {X 0,Y 481.668,Z 692.477,A -85,B 0,C 180,E1 -6980.059,E2 -6980.059} C_VEL
LIN {X 0,Y 481.62,Z 692.489,A -85,B 0,C 180,E1 -6983.252,E2 -6983.252} C_VEL
LIN {X 0,Y 481.699,Z 692.477,A -85,B 0,C 180,E1 -6986.329,E2 -6986.329} C_VEL
LIN {X 0,Y 481.648,Z 692.492,A -85,B 0,C 180,E1 -6989.415,E2 -6989.415} C_VEL
LIN {X 0,Y 481.692,Z 692.478,A -85,B 0,C 180,E1 -6992.168,E2 -6992.168} C_VEL
LIN {X 0,Y 481.707,Z 692.478,A -85,B 0,C 180,E1 -6994.969,E2 -6994.969} C_VEL
LIN {X 0,Y 481.639,Z 692.489,A -85,B 0,C 180,E1 -6997.704,E2 -6997.704} C_VEL
LIN {X 0,Y 481.694,Z 692.479,A -85,B 0,C 180,E1 -7000.393,E2 -7000.393} C_VEL
LIN {X 0,Y 481.678,Z 692.477,A -85,B 0,C 180,E1 -7003.034,E2 -7003.034} C_VEL
LIN {X 0,Y 481.678,Z 692.486,A -85,B 0,C 180,E1 -7005.638,E2 -7005.638} C_VEL
LIN {X 0,Y 481.738,Z 692.478,A -85,B 0,C 180,E1 -7008.215,E2 -7008.215} C_VEL
LIN {X 0,Y 481.751,Z 692.47,A -85,B 0,C 180,E1 -7011.612,E2 -7011.612} C_VEL
LIN {X 0,Y 481.797,Z 692.473,A -85,B 0,C 180,E1 -7014.139,E2 -7014.139} C_VEL
LIN {X 0,Y 481.916,Z 692.45,A -85,B 0,C 180,E1 -7017.493,E2 -7017.493} C_VEL
LIN {X 0,Y 481.894,Z 692.455,A -85,B 0,C 180,E1 -7020.836,E2 -7020.836} C_VEL
LIN {X 0,Y 481.915,Z 692.458,A -85,B 0,C 180,E1 -7022.508,E2 -7022.508} C_VEL
LIN {X 0,Y 481.797,Z 692.465,A -85,B 0,C 180,E1 -7025.861,E2 -7025.861} C_VEL
LIN {X 0,Y 481.752,Z 692.475,A -85,B 0,C 180,E1 -7028.389,E2 -7028.389} C_VEL
LIN {X 0,Y 481.741,Z 692.471,A -85,B 0,C 180,E1 -7031.785,E2 -7031.785} C_VEL
LIN {X 0,Y 481.73,Z 692.475,A -85,B 0,C 180,E1 -7035.225,E2 -7035.225} C_VEL
LIN {X 0,Y 481.697,Z 692.483,A -85,B 0,C 180,E1 -7038.723,E2 -7038.723} C_VEL
LIN {X 0,Y 481.634,Z 692.489,A -85,B 0,C 180,E1 -7041.396,E2 -7041.396} C_VEL
LIN {X 0,Y 481.64,Z 692.48,A -85,B 0,C 180,E1 -7044.115,E2 -7044.115} C_VEL
LIN {X 0,Y 481.704,Z 692.485,A -85,B 0,C 180,E1 -7047.133,E2 -7047.133} C_VEL
LIN {X 0,Y 481.668,Z 692.488,A -85,B 0,C 180,E1 -7049.742,E2 -7049.742} C_VEL
LIN {X 0,Y 481.663,Z 692.479,A -85,B 0,C 180,E1 -7052.675,E2 -7052.675} C_VEL
LIN {X 0,Y 481.633,Z 692.49,A -85,B 0,C 180,E1 -7055.71,E2 -7055.71} C_VEL
LIN {X 0,Y 481.662,Z 692.48,A -85,B 0,C 180,E1 -7058.86,E2 -7058.86} C_VEL
LIN {X 0,Y 481.645,Z 692.493,A -85,B 0,C 180,E1 -7061.914,E2 -7061.914} C_VEL
LIN {X 0,Y 481.648,Z 692.488,A -85,B 0,C 180,E1 -7064.459,E2 -7064.459} C_VEL
LIN {X 0,Y 481.637,Z 692.493,A -85,B 0,C 180,E1 -7067.84,E2 -7067.84} C_VEL
LIN {X 0,Y 481.705,Z 692.75,A -85,B 0,C 180,E1 -7068.821,E2 -7068.821} C_VEL
LIN {X 0,Y 481.971,Z 693.809,A -85,B 0,C 180,E1 -7068.941,E2 -7068.941} C_VEL
LIN {X 0,Y 485.131,Z 702.401,A -85,B 0,C 180,E1 -7069.195,E2 -7069.195} C_VEL
LIN {X 0,Y 484.631,Z 773.478,A -85,B 0,C 180,E1 -7070.29,E2 -7070.29} C_VEL
LIN {X 0,Y 484.533,Z 786.983,A -85,B 0,C 180,E1 -7070.68,E2 -7070.68} C_VEL
LIN {X 0,Y 484.364,Z 799.131,A -85,B 0,C 180,E1 -7071.199,E2 -7071.199} C_VEL
LIN {X 0,Y 484.14,Z 810.066,A -85,B 0,C 180,E1 -7071.825,E2 -7071.825} C_VEL
LIN {X 0,Y 483.774,Z 820.723,A -85,B 0,C 180,E1 -7072.601,E2 -7072.601} C_VEL
LIN {X 0,Y 483.404,Z 831.06,A -85,B 0,C 180,E1 -7073.542,E2 -7073.542} C_VEL
LIN {X 0,Y 483.294,Z 833.637,A -85,B 0,C 180,E1 -7073.808,E2 -7073.808} C_VEL
LIN {X 0,Y 482.457,Z 838.032,A -85,B 0,C 180,E1 -7074.277,E2 -7074.277} C_VEL
LIN {X 0,Y 479.32,Z 844.941,A -85,B 0,C 180,E1 -7075.042,E2 -7075.042} C_VEL
LIN {X 0,Y 476.215,Z 851.261,A -85,B 0,C 180,E1 -7075.872,E2 -7075.872} C_VEL
LIN {X 0,Y 475.427,Z 854.695,A -85,B 0,C 180,E1 -7076.436,E2 -7076.436} C_VEL
LIN {X 0,Y 475.083,Z 861.555,A -85,B 0,C 180,E1 -7077.823,E2 -7077.823} C_VEL
LIN {X 0,Y 474.833,Z 866.637,A -85,B 0,C 180,E1 -7079.145,E2 -7079.145} C_VEL
LIN {X 0,Y 474.643,Z 871.212,A -85,B 0,C 180,E1 -7080.751,E2 -7080.751} C_VEL
LIN {X 0,Y 474.514,Z 873.229,A -85,B 0,C 180,E1 -7081.711,E2 -7081.711} C_VEL
LIN {X 0,Y 474.468,Z 874.72,A -85,B 0,C 180,E1 -7082.717,E2 -7082.717} C_VEL
LIN {X 0,Y 474.409,Z 875.626,A -85,B 0,C 180,E1 -7083.615,E2 -7083.615} C_VEL
LIN {X 0,Y 474.365,Z 876.09,A -85,B 0,C 180,E1 -7084.657,E2 -7084.657} C_VEL
LIN {X 0,Y 474.358,Z 876.057,A -85,B 0,C 180,E1 -7085.492,E2 -7085.492} C_VEL
LIN {X 0,Y 474.358,Z 875.328,A -85,B 0,C 180,E1 -7086.721,E2 -7086.721} C_VEL
LIN {X 0,Y 474.484,Z 873.243,A -85,B 0,C 180,E1 -7088.268,E2 -7088.268} C_VEL
LIN {X 0,Y 474.644,Z 870.257,A -85,B 0,C 180,E1 -7089.639,E2 -7089.639} C_VEL
LIN {X 0,Y 474.843,Z 866.155,A -85,B 0,C 180,E1 -7090.999,E2 -7090.999} C_VEL
LIN {X 0,Y 475.084,Z 860.812,A -85,B 0,C 180,E1 -7092.348,E2 -7092.348} C_VEL
LIN {X 0,Y 475.36,Z 854.067,A -85,B 0,C 180,E1 -7093.687,E2 -7093.687} C_VEL
LIN {X 0,Y 475.803,Z 845.63,A -85,B 0,C 180,E1 -7095.021,E2 -7095.021} C_VEL
LIN {X 0,Y 476.161,Z 836.976,A -85,B 0,C 180,E1 -7096.124,E2 -7096.124} C_VEL
LIN {X 0,Y 476.624,Z 826.225,A -85,B 0,C 180,E1 -7097.223,E2 -7097.223} C_VEL
LIN {X 0,Y 477.027,Z 815.539,A -85,B 0,C 180,E1 -7098.098,E2 -7098.098} C_VEL
LIN {X 0,Y 477.348,Z 803.651,A -85,B 0,C 180,E1 -7098.859,E2 -7098.859} C_VEL
LIN {X 0,Y 477.622,Z 791.239,A -85,B 0,C 180,E1 -7099.456,E2 -7099.456} C_VEL
LIN {X 0,Y 477.739,Z 778.589,A -85,B 0,C 180,E1 -7099.887,E2 -7099.887} C_VEL
LIN {X 0,Y 477.792,Z 764.651,A -85,B 0,C 180,E1 -7100.167,E2 -7100.167} C_VEL
LIN {X 0,Y 478.159,Z 703.504,A -85,B 0,C 180,E1 -7101.097,E2 -7101.097} C_VEL
LIN {X 0,Y 474.934,Z 694.528,A -85,B 0,C 180,E1 -7101.371,E2 -7101.371} C_VEL
LIN {X 0,Y 474.715,Z 693.614,A -85,B 0,C 180,E1 -7101.488,E2 -7101.488} C_VEL
LIN {X 0,Y 474.723,Z 693.354,A -85,B 0,C 180,E1 -7102.344,E2 -7102.344} C_VEL
LIN {X 0,Y 474.732,Z 693.348,A -85,B 0,C 180,E1 -7104.905,E2 -7104.905} C_VEL
LIN {X 0,Y 474.874,Z 693.332,A -85,B 0,C 180,E1 -7107.457,E2 -7107.457} C_VEL
LIN {X 0,Y 474.883,Z 693.332,A -85,B 0,C 180,E1 -7110.001,E2 -7110.001} C_VEL
LIN {X 0,Y 474.873,Z 693.336,A -85,B 0,C 180,E1 -7112.546,E2 -7112.546} C_VEL
LIN {X 0,Y 474.74,Z 693.349,A -85,B 0,C 180,E1 -7115.949,E2 -7115.949} C_VEL
LIN {X 0,Y 474.665,Z 693.362,A -85,B 0,C 180,E1 -7118.516,E2 -7118.516} C_VEL
LIN {X 0,Y 474.689,Z 693.351,A -85,B 0,C 180,E1 -7121.964,E2 -7121.964} C_VEL
LIN {X 0,Y 474.703,Z 693.347,A -85,B 0,C 180,E1 -7125.457,E2 -7125.457} C_VEL
LIN {X 0,Y 474.615,Z 693.36,A -85,B 0,C 180,E1 -7129.014,E2 -7129.014} C_VEL
LIN {X 0,Y 474.591,Z 693.363,A -85,B 0,C 180,E1 -7131.73,E2 -7131.73} C_VEL
LIN {X 0,Y 474.625,Z 693.361,A -85,B 0,C 180,E1 -7134.496,E2 -7134.496} C_VEL
LIN {X 0,Y 474.599,Z 693.362,A -85,B 0,C 180,E1 -7137.327,E2 -7137.327} C_VEL
LIN {X 0,Y 474.555,Z 693.368,A -85,B 0,C 180,E1 -7140.235,E2 -7140.235} C_VEL
LIN {X 0,Y 474.605,Z 693.36,A -85,B 0,C 180,E1 -7143.224,E2 -7143.224} C_VEL
LIN {X 0,Y 474.571,Z 693.358,A -85,B 0,C 180,E1 -7146.326,E2 -7146.326} C_VEL
LIN {X 0,Y 474.602,Z 693.369,A -85,B 0,C 180,E1 -7149.551,E2 -7149.551} C_VEL
LIN {X 0,Y 474.571,Z 693.367,A -85,B 0,C 180,E1 -7152.941,E2 -7152.941} C_VEL
LIN {X 0,Y 474.586,Z 693.369,A -85,B 0,C 180,E1 -7155.892,E2 -7155.892} C_VEL
LIN {X 0,Y 474.586,Z 693.365,A -85,B 0,C 180,E1 -7159.048,E2 -7159.048} C_VEL
LIN {X 0,Y 474.586,Z 693.371,A -85,B 0,C 180,E1 -7161.709,E2 -7161.709} C_VEL
LIN {X 0,Y 474.584,Z 693.366,A -85,B 0,C 180,E1 -7164.722,E2 -7164.722} C_VEL
LIN {X 0,Y 474.616,Z 693.368,A -85,B 0,C 180,E1 -7167.786,E2 -7167.786} C_VEL
LIN {X 0,Y 474.624,Z 693.531,A -85,B 0,C 180,E1 -7170.718,E2 -7170.718} C_VEL
LIN {X 0,Y 474.876,Z 694.623,A -85,B 0,C 180,E1 -7170.864,E2 -7170.864} C_VEL
LIN {X 0,Y 477.928,Z 703.361,A -85,B 0,C 180,E1 -7171.123,E2 -7171.123} C_VEL
LIN {X 0,Y 477.343,Z 768.59,A -85,B 0,C 180,E1 -7172.168,E2 -7172.168} C_VEL
LIN {X 0,Y 477.206,Z 780.26,A -85,B 0,C 180,E1 -7172.484,E2 -7172.484} C_VEL
LIN {X 0,Y 477.032,Z 790.599,A -85,B 0,C 180,E1 -7172.884,E2 -7172.884} C_VEL
LIN {X 0,Y 476.779,Z 800.821,A -85,B 0,C 180,E1 -7173.401,E2 -7173.401} C_VEL
LIN {X 0,Y 476.454,Z 810.73,A -85,B 0,C 180,E1 -7174.032,E2 -7174.032} C_VEL
LIN {X 0,Y 476.148,Z 820.158,A -85,B 0,C 180,E1 -7174.773,E2 -7174.773} C_VEL
LIN {X 0,Y 475.772,Z 828.587,A -85,B 0,C 180,E1 -7175.568,E2 -7175.568} C_VEL
LIN {X 0,Y 475.504,Z 836.646,A -85,B 0,C 180,E1 -7176.48,E2 -7176.48} C_VEL
LIN {X 0,Y 475.231,Z 843.457,A -85,B 0,C 180,E1 -7177.387,E2 -7177.387} C_VEL
LIN {X 0,Y 474.853,Z 851.102,A -85,B 0,C 180,E1 -7178.627,E2 -7178.627} C_VEL
LIN {X 0,Y 474.636,Z 856.281,A -85,B 0,C 180,E1 -7179.637,E2 -7179.637} C_VEL
LIN {X 0,Y 474.522,Z 860.197,A -85,B 0,C 180,E1 -7180.534,E2 -7180.534} C_VEL
LIN {X 0,Y 474.359,Z 864.867,A -85,B 0,C 180,E1 -7181.872,E2 -7181.872} C_VEL
LIN {X 0,Y 474.244,Z 867.24,A -85,B 0,C 180,E1 -7182.759,E2 -7182.759} C_VEL
LIN {X 0,Y 474.143,Z 870.727,A -85,B 0,C 180,E1 -7184.526,E2 -7184.526} C_VEL
LIN {X 0,Y 474.098,Z 872.414,A -85,B 0,C 180,E1 -7186.279,E2 -7186.279} C_VEL
LIN {X 0,Y 474.104,Z 872.607,A -85,B 0,C 180,E1 -7187.152,E2 -7187.152} C_VEL
LIN {X 0,Y 474.139,Z 872.367,A -85,B 0,C 180,E1 -7188.045,E2 -7188.045} C_VEL
LIN {X 0,Y 474.222,Z 870.717,A -85,B 0,C 180,E1 -7189.756,E2 -7189.756} C_VEL
LIN {X 0,Y 474.331,Z 867.268,A -85,B 0,C 180,E1 -7191.479,E2 -7191.479} C_VEL
LIN {X 0,Y 474.476,Z 864.985,A -85,B 0,C 180,E1 -7192.339,E2 -7192.339} C_VEL
LIN {X 0,Y 474.663,Z 860.511,A -85,B 0,C 180,E1 -7193.624,E2 -7193.624} C_VEL
LIN {X 0,Y 474.814,Z 854.824,A -85,B 0,C 180,E1 -7194.905,E2 -7194.905} C_VEL
LIN {X 0,Y 475.046,Z 849.035,A -85,B 0,C 180,E1 -7195.97,E2 -7195.97} C_VEL
LIN {X 0,Y 475.41,Z 842.022,A -85,B 0,C 180,E1 -7197.034,E2 -7197.034} C_VEL
LIN {X 0,Y 475.744,Z 833.532,A -85,B 0,C 180,E1 -7198.095,E2 -7198.095} C_VEL
LIN {X 0,Y 476.085,Z 825.361,A -85,B 0,C 180,E1 -7198.943,E2 -7198.943} C_VEL
LIN {X 0,Y 476.397,Z 816.832,A -85,B 0,C 180,E1 -7199.683,E2 -7199.683} C_VEL
LIN {X 0,Y 476.682,Z 808.06,A -85,B 0,C 180,E1 -7200.317,E2 -7200.317} C_VEL
LIN {X 0,Y 476.935,Z 798.127,A -85,B 0,C 180,E1 -7200.897,E2 -7200.897} C_VEL
LIN {X 0,Y 477.181,Z 786.94,A -85,B 0,C 180,E1 -7201.398,E2 -7201.398} C_VEL
LIN {X 0,Y 477.295,Z 776.551,A -85,B 0,C 180,E1 -7201.74,E2 -7201.74} C_VEL
LIN {X 0,Y 477.37,Z 764.529,A -85,B 0,C 180,E1 -7202.004,E2 -7202.004} C_VEL
LIN {X 0,Y 477.848,Z 702.44,A -85,B 0,C 180,E1 -7203.003,E2 -7203.003} C_VEL
LIN {X 0,Y 474.953,Z 694.514,A -85,B 0,C 180,E1 -7203.26,E2 -7203.26} C_VEL
LIN {X 0,Y 474.704,Z 693.479,A -85,B 0,C 180,E1 -7203.421,E2 -7203.421} C_VEL
LIN {X 0,Y 474.764,Z 693.35,A -85,B 0,C 180,E1 -7205.948,E2 -7205.948} C_VEL
LIN {X 0,Y 474.718,Z 693.353,A -85,B 0,C 180,E1 -7208.514,E2 -7208.514} C_VEL
LIN {X 0,Y 474.712,Z 693.353,A -85,B 0,C 180,E1 -7211.962,E2 -7211.962} C_VEL
LIN {X 0,Y 474.707,Z 693.35,A -85,B 0,C 180,E1 -7215.455,E2 -7215.455} C_VEL
LIN {X 0,Y 474.67,Z 693.357,A -85,B 0,C 180,E1 -7219.01,E2 -7219.01} C_VEL
LIN {X 0,Y 474.595,Z 693.364,A -85,B 0,C 180,E1 -7221.729,E2 -7221.729} C_VEL
LIN {X 0,Y 474.647,Z 693.363,A -85,B 0,C 180,E1 -7224.493,E2 -7224.493} C_VEL
LIN {X 0,Y 474.644,Z 693.36,A -85,B 0,C 180,E1 -7227.323,E2 -7227.323} C_VEL
LIN {X 0,Y 474.61,Z 693.364,A -85,B 0,C 180,E1 -7230.23,E2 -7230.23} C_VEL
LIN {X 0,Y 474.631,Z 693.364,A -85,B 0,C 180,E1 -7233.221,E2 -7233.221} C_VEL
LIN {X 0,Y 474.595,Z 693.364,A -85,B 0,C 180,E1 -7236.323,E2 -7236.323} C_VEL
LIN {X 0,Y 474.634,Z 693.361,A -85,B 0,C 180,E1 -7239.647,E2 -7239.647} C_VEL
LIN {X 0,Y 474.621,Z 693.365,A -85,B 0,C 180,E1 -7242.934,E2 -7242.934} C_VEL
LIN {X 0,Y 474.611,Z 693.364,A -85,B 0,C 180,E1 -7245.894,E2 -7245.894} C_VEL
LIN {X 0,Y 474.634,Z 693.362,A -85,B 0,C 180,E1 -7249.04,E2 -7249.04} C_VEL
LIN {X 0,Y 474.612,Z 693.368,A -85,B 0,C 180,E1 -7251.704,E2 -7251.704} C_VEL
LIN {X 0,Y 474.626,Z 693.362,A -85,B 0,C 180,E1 -7254.725,E2 -7254.725} C_VEL
LIN {X 0,Y 474.641,Z 693.365,A -85,B 0,C 180,E1 -7257.787,E2 -7257.787} C_VEL
LIN {X 0,Y 474.682,Z 693.529,A -85,B 0,C 180,E1 -7259.555,E2 -7259.555} C_VEL
LIN {X 0,Y 478.293,Z 709.354,A -85,B 0,C 180,E1 -7261.951,E2 -7261.951} C_VEL
LIN {X 0,Y 478.813,Z 712.917,A -85,B 0,C 180,E1 -7262.46,E2 -7262.46} C_VEL
LIN {X 0,Y 477.665,Z 737.188,A -85,B 0,C 180,E1 -7265.67,E2 -7265.67} C_VEL
LIN {X 0,Y 476.823,Z 759.7,A -85,B 0,C 180,E1 -7268.604,E2 -7268.604} C_VEL
LIN {X 0,Y 475.923,Z 785.604,A -85,B 0,C 180,E1 -7271.933,E2 -7271.933} C_VEL
LIN {X 0,Y 475.613,Z 795.802,A -85,B 0,C 180,E1 -7273.208,E2 -7273.208} C_VEL
LIN {X 0,Y 477.93,Z 817.104,A -85,B 0,C 180,E1 -7273.631,E2 -7273.631} C_VEL
LIN {X 0,Y 477.296,Z 906.906,A -85,B 0,C 180,E1 -7275.012,E2 -7275.012} C_VEL
LIN {X 0,Y 476.878,Z 920.771,A -85,B 0,C 180,E1 -7275.408,E2 -7275.408} C_VEL
LIN {X 0,Y 476.438,Z 933.768,A -85,B 0,C 180,E1 -7275.966,E2 -7275.966} C_VEL
LIN {X 0,Y 475.98,Z 945.642,A -85,B 0,C 180,E1 -7276.66,E2 -7276.66} C_VEL
LIN {X 0,Y 475.547,Z 957.364,A -85,B 0,C 180,E1 -7277.536,E2 -7277.536} C_VEL
LIN {X 0,Y 475.019,Z 967.493,A -85,B 0,C 180,E1 -7278.477,E2 -7278.477} C_VEL
LIN {X 0,Y 474.681,Z 976.853,A -85,B 0,C 180,E1 -7279.549,E2 -7279.549} C_VEL
LIN {X 0,Y 474.37,Z 985.984,A -85,B 0,C 180,E1 -7280.834,E2 -7280.834} C_VEL
LIN {X 0,Y 474.145,Z 993.351,A -85,B 0,C 180,E1 -7282.118,E2 -7282.118} C_VEL
LIN {X 0,Y 474.007,Z 999.294,A -85,B 0,C 180,E1 -7283.412,E2 -7283.412} C_VEL
LIN {X 0,Y 473.979,Z 1003.19,A -85,B 0,C 180,E1 -7284.468,E2 -7284.468} C_VEL
LIN {X 0,Y 473.925,Z 1006.899,A -85,B 0,C 180,E1 -7285.747,E2 -7285.747} C_VEL
LIN {X 0,Y 473.94,Z 1008.817,A -85,B 0,C 180,E1 -7286.598,E2 -7286.598} C_VEL
LIN {X 0,Y 473.898,Z 1010.249,A -85,B 0,C 180,E1 -7287.449,E2 -7287.449} C_VEL
LIN {X 0,Y 473.881,Z 1011.27,A -85,B 0,C 180,E1 -7288.299,E2 -7288.299} C_VEL
LIN {X 0,Y 473.853,Z 1011.886,A -85,B 0,C 180,E1 -7289.149,E2 -7289.149} C_VEL
LIN {X 0,Y 473.85,Z 1012.102,A -85,B 0,C 180,E1 -7289.999,E2 -7289.999} C_VEL
LIN {X 0,Y 473.855,Z 1011.874,A -85,B 0,C 180,E1 -7290.849,E2 -7290.849} C_VEL
LIN {X 0,Y 473.885,Z 1011.246,A -85,B 0,C 180,E1 -7291.698,E2 -7291.698} C_VEL
LIN {X 0,Y 473.903,Z 1010.212,A -85,B 0,C 180,E1 -7292.549,E2 -7292.549} C_VEL
LIN {X 0,Y 473.939,Z 1008.766,A -85,B 0,C 180,E1 -7293.399,E2 -7293.399} C_VEL
LIN {X 0,Y 473.932,Z 1005.724,A -85,B 0,C 180,E1 -7294.677,E2 -7294.677} C_VEL
LIN {X 0,Y 474.019,Z 1001.623,A -85,B 0,C 180,E1 -7295.956,E2 -7295.956} C_VEL
LIN {X 0,Y 474.097,Z 995.317,A -85,B 0,C 180,E1 -7297.451,E2 -7297.451} C_VEL
LIN {X 0,Y 474.299,Z 988.452,A -85,B 0,C 180,E1 -7298.735,E2 -7298.735} C_VEL
LIN {X 0,Y 474.553,Z 979.949,A -85,B 0,C 180,E1 -7300.02,E2 -7300.02} C_VEL
LIN {X 0,Y 474.921,Z 971.261,A -85,B 0,C 180,E1 -7301.09,E2 -7301.09} C_VEL
LIN {X 0,Y 475.39,Z 960.868,A -85,B 0,C 180,E1 -7302.132,E2 -7302.132} C_VEL
LIN {X 0,Y 475.806,Z 949.99,A -85,B 0,C 180,E1 -7303.016,E2 -7303.016} C_VEL
LIN {X 0,Y 476.179,Z 938.417,A -85,B 0,C 180,E1 -7303.767,E2 -7303.767} C_VEL
LIN {X 0,Y 476.692,Z 926.563,A -85,B 0,C 180,E1 -7304.35,E2 -7304.35} C_VEL
LIN {X 0,Y 477.094,Z 912.932,A -85,B 0,C 180,E1 -7304.828,E2 -7304.828} C_VEL
LIN {X 0,Y 477.369,Z 899.327,A -85,B 0,C 180,E1 -7305.12,E2 -7305.12} C_VEL
LIN {X 0,Y 477.88,Z 815.464,A -85,B 0,C 180,E1 -7306.387,E2 -7306.387} C_VEL
LIN {X 0,Y 475.57,Z 795.046,A -85,B 0,C 180,E1 -7306.803,E2 -7306.803} C_VEL
LIN {X 0,Y 476.253,Z 772.64,A -85,B 0,C 180,E1 -7309.634,E2 -7309.634} C_VEL
LIN {X 0,Y 477.169,Z 748.482,A -85,B 0,C 180,E1 -7312.743,E2 -7312.743} C_VEL
LIN {X 0,Y 478.147,Z 722.387,A -85,B 0,C 180,E1 -7316.163,E2 -7316.163} C_VEL
LIN {X 0,Y 478.562,Z 710.697,A -85,B 0,C 180,E1 -7317.725,E2 -7317.725} C_VEL
LIN {X 0,Y 474.688,Z 693.62,A -85,B 0,C 180,E1 -7320.295,E2 -7320.295} C_VEL
LIN {X 0,Y 474.594,Z 693.365,A -85,B 0,C 180,E1 -7321.216,E2 -7321.216} C_VEL
LIN {X 0,Y 474.626,Z 693.359,A -85,B 0,C 180,E1 -7324.24,E2 -7324.24} C_VEL
LIN {X 0,Y 474.583,Z 693.367,A -85,B 0,C 180,E1 -7327.382,E2 -7327.382} C_VEL
LIN {X 0,Y 474.62,Z 693.362,A -85,B 0,C 180,E1 -7329.646,E2 -7329.646} C_VEL
LIN {X 0,Y 474.607,Z 693.364,A -85,B 0,C 180,E1 -7332.933,E2 -7332.933} C_VEL
LIN {X 0,Y 474.61,Z 693.359,A -85,B 0,C 180,E1 -7335.895,E2 -7335.895} C_VEL
LIN {X 0,Y 474.624,Z 693.361,A -85,B 0,C 180,E1 -7339.039,E2 -7339.039} C_VEL
LIN {X 0,Y 474.602,Z 693.363,A -85,B 0,C 180,E1 -7341.703,E2 -7341.703} C_VEL
LIN {X 0,Y 474.62,Z 693.357,A -85,B 0,C 180,E1 -7344.725,E2 -7344.725} C_VEL
LIN {X 0,Y 474.626,Z 693.36,A -85,B 0,C 180,E1 -7347.787,E2 -7347.787} C_VEL
LIN {X 0,Y 474.622,Z 693.363,A -85,B 0,C 180,E1 -7350.882,E2 -7350.882} C_VEL
LIN {X 0,Y 474.656,Z 693.36,A -85,B 0,C 180,E1 -7353.628,E2 -7353.628} C_VEL
LIN {X 0,Y 474.624,Z 693.359,A -85,B 0,C 180,E1 -7356.641,E2 -7356.641} C_VEL
LIN {X 0,Y 474.643,Z 693.36,A -85,B 0,C 180,E1 -7360.089,E2 -7360.089} C_VEL
LIN {X 0,Y 474.638,Z 693.353,A -85,B 0,C 180,E1 -7362.774,E2 -7362.774} C_VEL
LIN {X 0,Y 474.636,Z 693.361,A -85,B 0,C 180,E1 -7365.421,E2 -7365.421} C_VEL
LIN {X 0,Y 474.692,Z 693.358,A -85,B 0,C 180,E1 -7368.037,E2 -7368.037} C_VEL
LIN {X 0,Y 474.716,Z 693.345,A -85,B 0,C 180,E1 -7371.486,E2 -7371.486} C_VEL
LIN {X 0,Y 474.759,Z 693.35,A -85,B 0,C 180,E1 -7374.052,E2 -7374.052} C_VEL
LIN {X 0,Y 474.882,Z 693.326,A -85,B 0,C 180,E1 -7377.455,E2 -7377.455} C_VEL
LIN {X 0,Y 474.846,Z 693.333,A -85,B 0,C 180,E1 -7380.848,E2 -7380.848} C_VEL
LIN {X 0,Y 474.882,Z 693.334,A -85,B 0,C 180,E1 -7382.545,E2 -7382.545} C_VEL
LIN {X 0,Y 474.759,Z 693.342,A -85,B 0,C 180,E1 -7385.948,E2 -7385.948} C_VEL
LIN {X 0,Y 474.717,Z 693.352,A -85,B 0,C 180,E1 -7388.514,E2 -7388.514} C_VEL
LIN {X 0,Y 474.694,Z 693.349,A -85,B 0,C 180,E1 -7391.963,E2 -7391.963} C_VEL
LIN {X 0,Y 474.688,Z 693.35,A -85,B 0,C 180,E1 -7395.456,E2 -7395.456} C_VEL
LIN {X 0,Y 474.651,Z 693.361,A -85,B 0,C 180,E1 -7399.011,E2 -7399.011} C_VEL
LIN {X 0,Y 474.577,Z 693.365,A -85,B 0,C 180,E1 -7401.73,E2 -7401.73} C_VEL
LIN {X 0,Y 474.619,Z 693.355,A -85,B 0,C 180,E1 -7404.495,E2 -7404.495} C_VEL
LIN {X 0,Y 474.663,Z 693.358,A -85,B 0,C 180,E1 -7407.333,E2 -7407.333} C_VEL
LIN {X 0,Y 474.595,Z 693.365,A -85,B 0,C 180,E1 -7410.231,E2 -7410.231} C_VEL
LIN {X 0,Y 474.634,Z 693.358,A -85,B 0,C 180,E1 -7413.221,E2 -7413.221} C_VEL
LIN {X 0,Y 474.583,Z 693.366,A -85,B 0,C 180,E1 -7416.324,E2 -7416.324} C_VEL
LIN {X 0,Y 474.619,Z 693.365,A -85,B 0,C 180,E1 -7419.649,E2 -7419.649} C_VEL
LIN {X 0,Y 474.607,Z 693.362,A -85,B 0,C 180,E1 -7422.936,E2 -7422.936} C_VEL
LIN {X 0,Y 474.597,Z 693.367,A -85,B 0,C 180,E1 -7425.896,E2 -7425.896} C_VEL
LIN {X 0,Y 474.626,Z 693.557,A -85,B 0,C 180,E1 -7428.544,E2 -7428.544} C_VEL
LIN {X 0,Y 474.925,Z 694.706,A -85,B 0,C 180,E1 -7428.689,E2 -7428.689} C_VEL
LIN {X 0,Y 478.333,Z 704.035,A -85,B 0,C 180,E1 -7428.972,E2 -7428.972} C_VEL
LIN {X 0,Y 477.841,Z 774.293,A -85,B 0,C 180,E1 -7430.069,E2 -7430.069} C_VEL
LIN {X 0,Y 477.739,Z 787.126,A -85,B 0,C 180,E1 -7430.438,E2 -7430.438} C_VEL
LIN {X 0,Y 477.586,Z 798.418,A -85,B 0,C 180,E1 -7430.912,E2 -7430.912} C_VEL
LIN {X 0,Y 477.33,Z 809.531,A -85,B 0,C 180,E1 -7431.531,E2 -7431.531} C_VEL
LIN {X 0,Y 476.987,Z 820.417,A -85,B 0,C 180,E1 -7432.307,E2 -7432.307} C_VEL
LIN {X 0,Y 476.597,Z 830.395,A -85,B 0,C 180,E1 -7433.199,E2 -7433.199} C_VEL
LIN {X 0,Y 476.166,Z 840.086,A -85,B 0,C 180,E1 -7434.271,E2 -7434.271} C_VEL
LIN {X 0,Y 475.731,Z 847.996,A -85,B 0,C 180,E1 -7435.338,E2 -7435.338} C_VEL
LIN {X 0,Y 475.427,Z 854.695,A -85,B 0,C 180,E1 -7436.436,E2 -7436.436} C_VEL
LIN {X 0,Y 474.648,Z 857.96,A -85,B 0,C 180,E1 -7437.023,E2 -7437.023} C_VEL
LIN {X 0,Y 471.571,Z 862.975,A -85,B 0,C 180,E1 -7437.991,E2 -7437.991} C_VEL
LIN {X 0,Y 468.501,Z 867.4,A -85,B 0,C 180,E1 -7439.011,E2 -7439.011} C_VEL
LIN {X 0,Y 467.745,Z 869.577,A -85,B 0,C 180,E1 -7439.674,E2 -7439.674} C_VEL
LIN {X 0,Y 467.64,Z 872.159,A -85,B 0,C 180,E1 -7440.653,E2 -7440.653} C_VEL
LIN {X 0,Y 467.453,Z 875.151,A -85,B 0,C 180,E1 -7442.222,E2 -7442.222} C_VEL
LIN {X 0,Y 467.424,Z 876.287,A -85,B 0,C 180,E1 -7443.189,E2 -7443.189} C_VEL
LIN {X 0,Y 467.365,Z 877.07,A -85,B 0,C 180,E1 -7444.456,E2 -7444.456} C_VEL
LIN {X 0,Y 467.344,Z 876.84,A -85,B 0,C 180,E1 -7446.046,E2 -7446.046} C_VEL
LIN {X 0,Y 467.344,Z 876.109,A -85,B 0,C 180,E1 -7446.985,E2 -7446.985} C_VEL
LIN {X 0,Y 467.445,Z 874.894,A -85,B 0,C 180,E1 -7447.923,E2 -7447.923} C_VEL
LIN {X 0,Y 467.612,Z 872.189,A -85,B 0,C 180,E1 -7449.319,E2 -7449.319} C_VEL
LIN {X 0,Y 467.789,Z 868.394,A -85,B 0,C 180,E1 -7450.701,E2 -7450.701} C_VEL
LIN {X 0,Y 468.04,Z 863.4,A -85,B 0,C 180,E1 -7452.073,E2 -7452.073} C_VEL
LIN {X 0,Y 468.31,Z 857.095,A -85,B 0,C 180,E1 -7453.434,E2 -7453.434} C_VEL
LIN {X 0,Y 468.671,Z 850.595,A -85,B 0,C 180,E1 -7454.565,E2 -7454.565} C_VEL
LIN {X 0,Y 469.058,Z 842.784,A -85,B 0,C 180,E1 -7455.688,E2 -7455.688} C_VEL
LIN {X 0,Y 469.507,Z 832.734,A -85,B 0,C 180,E1 -7456.857,E2 -7456.857} C_VEL
LIN {X 0,Y 469.936,Z 822.585,A -85,B 0,C 180,E1 -7457.806,E2 -7457.806} C_VEL
LIN {X 0,Y 470.358,Z 810.687,A -85,B 0,C 180,E1 -7458.692,E2 -7458.692} C_VEL
LIN {X 0,Y 470.657,Z 797.981,A -85,B 0,C 180,E1 -7459.407,E2 -7459.407} C_VEL
LIN {X 0,Y 470.832,Z 785.069,A -85,B 0,C 180,E1 -7459.936,E2 -7459.936} C_VEL
LIN {X 0,Y 470.953,Z 771.835,A -85,B 0,C 180,E1 -7460.28,E2 -7460.28} C_VEL
LIN {X 0,Y 471.296,Z 704.883,A -85,B 0,C 180,E1 -7461.328,E2 -7461.328} C_VEL
LIN {X 0,Y 467.851,Z 695.279,A -85,B 0,C 180,E1 -7461.626,E2 -7461.626} C_VEL
LIN {X 0,Y 467.683,Z 694.323,A -85,B 0,C 180,E1 -7461.794,E2 -7461.794} C_VEL
LIN {X 0,Y 467.704,Z 694.224,A -85,B 0,C 180,E1 -7464.829,E2 -7464.829} C_VEL
LIN {X 0,Y 467.814,Z 694.211,A -85,B 0,C 180,E1 -7467.418,E2 -7467.418} C_VEL
LIN {X 0,Y 467.852,Z 694.208,A -85,B 0,C 180,E1 -7470.001,E2 -7470.001} C_VEL
LIN {X 0,Y 467.813,Z 694.215,A -85,B 0,C 180,E1 -7472.584,E2 -7472.584} C_VEL
LIN {X 0,Y 467.705,Z 694.226,A -85,B 0,C 180,E1 -7476.039,E2 -7476.039} C_VEL
LIN {X 0,Y 467.634,Z 694.237,A -85,B 0,C 180,E1 -7478.645,E2 -7478.645} C_VEL
LIN {X 0,Y 467.648,Z 694.232,A -85,B 0,C 180,E1 -7482.351,E2 -7482.351} C_VEL
LIN {X 0,Y 467.63,Z 694.228,A -85,B 0,C 180,E1 -7485.875,E2 -7485.875} C_VEL
LIN {X 0,Y 467.563,Z 694.234,A -85,B 0,C 180,E1 -7489.312,E2 -7489.312} C_VEL
LIN {X 0,Y 467.535,Z 694.241,A -85,B 0,C 180,E1 -7492.075,E2 -7492.075} C_VEL
LIN {X 0,Y 467.551,Z 694.244,A -85,B 0,C 180,E1 -7494.892,E2 -7494.892} C_VEL
LIN {X 0,Y 467.543,Z 694.238,A -85,B 0,C 180,E1 -7497.775,E2 -7497.775} C_VEL
LIN {X 0,Y 467.533,Z 694.249,A -85,B 0,C 180,E1 -7501.037,E2 -7501.037} C_VEL
LIN {X 0,Y 467.568,Z 694.226,A -85,B 0,C 180,E1 -7504.238,E2 -7504.238} C_VEL
LIN {X 0,Y 467.516,Z 694.242,A -85,B 0,C 180,E1 -7507.18,E2 -7507.18} C_VEL
LIN {X 0,Y 467.523,Z 694.244,A -85,B 0,C 180,E1 -7510.272,E2 -7510.272} C_VEL
LIN {X 0,Y 467.523,Z 694.244,A -85,B 0,C 180,E1 -7512.569,E2 -7512.569} C_VEL
LIN {X 0,Y 467.561,Z 694.241,A -85,B 0,C 180,E1 -7515.051,E2 -7515.051} C_VEL
LIN {X 0,Y 467.556,Z 694.24,A -85,B 0,C 180,E1 -7518.728,E2 -7518.728} C_VEL
LIN {X 0,Y 467.537,Z 694.249,A -85,B 0,C 180,E1 -7521.952,E2 -7521.952} C_VEL
LIN {X 0,Y 467.529,Z 694.245,A -85,B 0,C 180,E1 -7525.164,E2 -7525.164} C_VEL
LIN {X 0,Y 467.549,Z 694.249,A -85,B 0,C 180,E1 -7528.257,E2 -7528.257} C_VEL
LIN {X 0,Y 467.569,Z 694.397,A -85,B 0,C 180,E1 -7530.475,E2 -7530.475} C_VEL
LIN {X 0,Y 467.791,Z 695.349,A -85,B 0,C 180,E1 -7530.621,E2 -7530.621} C_VEL
LIN {X 0,Y 471.102,Z 704.829,A -85,B 0,C 180,E1 -7530.912,E2 -7530.912} C_VEL
LIN {X 0,Y 470.453,Z 770.346,A -85,B 0,C 180,E1 -7531.991,E2 -7531.991} C_VEL
LIN {X 0,Y 470.358,Z 781.344,A -85,B 0,C 180,E1 -7532.299,E2 -7532.299} C_VEL
LIN {X 0,Y 470.143,Z 791.463,A -85,B 0,C 180,E1 -7532.694,E2 -7532.694} C_VEL
LIN {X 0,Y 469.89,Z 801.708,A -85,B 0,C 180,E1 -7533.219,E2 -7533.219} C_VEL
LIN {X 0,Y 469.548,Z 812.224,A -85,B 0,C 180,E1 -7533.905,E2 -7533.905} C_VEL
LIN {X 0,Y 469.236,Z 821.08,A -85,B 0,C 180,E1 -7534.613,E2 -7534.613} C_VEL
LIN {X 0,Y 468.843,Z 829.527,A -85,B 0,C 180,E1 -7535.419,E2 -7535.419} C_VEL
LIN {X 0,Y 468.562,Z 837.402,A -85,B 0,C 180,E1 -7536.318,E2 -7536.318} C_VEL
LIN {X 0,Y 468.276,Z 844.432,A -85,B 0,C 180,E1 -7537.265,E2 -7537.265} C_VEL
LIN {X 0,Y 467.929,Z 851.464,A -85,B 0,C 180,E1 -7538.406,E2 -7538.406} C_VEL
LIN {X 0,Y 467.7,Z 856.279,A -85,B 0,C 180,E1 -7539.321,E2 -7539.321} C_VEL
LIN {X 0,Y 467.507,Z 862.042,A -85,B 0,C 180,E1 -7540.687,E2 -7540.687} C_VEL
LIN {X 0,Y 467.333,Z 866.485,A -85,B 0,C 180,E1 -7542.044,E2 -7542.044} C_VEL
LIN {X 0,Y 467.167,Z 869.774,A -85,B 0,C 180,E1 -7543.391,E2 -7543.391} C_VEL
LIN {X 0,Y 467.129,Z 871.541,A -85,B 0,C 180,E1 -7544.344,E2 -7544.344} C_VEL
LIN {X 0,Y 467.063,Z 873.314,A -85,B 0,C 180,E1 -7546.069,E2 -7546.069} C_VEL
LIN {X 0,Y 467.083,Z 873.638,A -85,B 0,C 180,E1 -7546.956,E2 -7546.956} C_VEL
LIN {X 0,Y 467.112,Z 873.456,A -85,B 0,C 180,E1 -7547.954,E2 -7547.954} C_VEL
LIN {X 0,Y 467.224,Z 872.03,A -85,B 0,C 180,E1 -7549.601,E2 -7549.601} C_VEL
LIN {X 0,Y 467.316,Z 868.81,A -85,B 0,C 180,E1 -7551.35,E2 -7551.35} C_VEL
LIN {X 0,Y 467.479,Z 866.612,A -85,B 0,C 180,E1 -7552.224,E2 -7552.224} C_VEL
LIN {X 0,Y 467.672,Z 862.331,A -85,B 0,C 180,E1 -7553.528,E2 -7553.528} C_VEL
LIN {X 0,Y 467.854,Z 855.745,A -85,B 0,C 180,E1 -7555.045,E2 -7555.045} C_VEL
LIN {X 0,Y 468.136,Z 849.907,A -85,B 0,C 180,E1 -7556.126,E2 -7556.126} C_VEL
LIN {X 0,Y 468.506,Z 842.851,A -85,B 0,C 180,E1 -7557.205,E2 -7557.205} C_VEL
LIN {X 0,Y 468.78,Z 836.228,A -85,B 0,C 180,E1 -7558.067,E2 -7558.067} C_VEL
LIN {X 0,Y 469.167,Z 827.216,A -85,B 0,C 180,E1 -7559.034,E2 -7559.034} C_VEL
LIN {X 0,Y 469.549,Z 817.437,A -85,B 0,C 180,E1 -7559.893,E2 -7559.893} C_VEL
LIN {X 0,Y 469.829,Z 808.552,A -85,B 0,C 180,E1 -7560.536,E2 -7560.536} C_VEL
LIN {X 0,Y 470.095,Z 798.447,A -85,B 0,C 180,E1 -7561.124,E2 -7561.124} C_VEL
LIN {X 0,Y 470.342,Z 787.724,A -85,B 0,C 180,E1 -7561.605,E2 -7561.605} C_VEL
LIN {X 0,Y 470.439,Z 777.253,A -85,B 0,C 180,E1 -7561.953,E2 -7561.953} C_VEL
LIN {X 0,Y 470.523,Z 765.078,A -85,B 0,C 180,E1 -7562.22,E2 -7562.22} C_VEL
LIN {X 0,Y 471.049,Z 703.736,A -85,B 0,C 180,E1 -7563.234,E2 -7563.234} C_VEL
LIN {X 0,Y 467.871,Z 695.327,A -85,B 0,C 180,E1 -7563.525,E2 -7563.525} C_VEL
LIN {X 0,Y 467.646,Z 694.35,A -85,B 0,C 180,E1 -7563.689,E2 -7563.689} C_VEL
LIN {X 0,Y 467.727,Z 694.226,A -85,B 0,C 180,E1 -7566.037,E2 -7566.037} C_VEL
LIN {X 0,Y 467.676,Z 694.23,A -85,B 0,C 180,E1 -7568.643,E2 -7568.643} C_VEL
LIN {X 0,Y 467.663,Z 694.232,A -85,B 0,C 180,E1 -7572.145,E2 -7572.145} C_VEL
LIN {X 0,Y 467.646,Z 694.231,A -85,B 0,C 180,E1 -7575.695,E2 -7575.695} C_VEL
LIN {X 0,Y 467.629,Z 694.233,A -85,B 0,C 180,E1 -7579.307,E2 -7579.307} C_VEL
LIN {X 0,Y 467.542,Z 694.245,A -85,B 0,C 180,E1 -7582.073,E2 -7582.073} C_VEL
LIN {X 0,Y 467.592,Z 694.241,A -85,B 0,C 180,E1 -7584.888,E2 -7584.888} C_VEL
LIN {X 0,Y 467.587,Z 694.237,A -85,B 0,C 180,E1 -7587.771,E2 -7587.771} C_VEL
LIN {X 0,Y 467.575,Z 694.245,A -85,B 0,C 180,E1 -7591.044,E2 -7591.044} C_VEL
LIN {X 0,Y 467.583,Z 694.238,A -85,B 0,C 180,E1 -7594.24,E2 -7594.24} C_VEL
LIN {X 0,Y 467.554,Z 694.247,A -85,B 0,C 180,E1 -7597.186,E2 -7597.186} C_VEL
LIN {X 0,Y 467.584,Z 694.237,A -85,B 0,C 180,E1 -7600.264,E2 -7600.264} C_VEL
LIN {X 0,Y 467.593,Z 694.237,A -85,B 0,C 180,E1 -7602.566,E2 -7602.566} C_VEL
LIN {X 0,Y 467.572,Z 694.243,A -85,B 0,C 180,E1 -7605.052,E2 -7605.052} C_VEL
LIN {X 0,Y 467.595,Z 694.242,A -85,B 0,C 180,E1 -7607.439,E2 -7607.439} C_VEL
LIN {X 0,Y 467.563,Z 694.24,A -85,B 0,C 180,E1 -7610.852,E2 -7610.852} C_VEL
LIN {X 0,Y 467.563,Z 694.242,A -85,B 0,C 180,E1 -7614.261,E2 -7614.261} C_VEL
LIN {X 0,Y 467.585,Z 694.241,A -85,B 0,C 180,E1 -7617.321,E2 -7617.321} C_VEL
LIN {X 0,Y 467.621,Z 694.465,A -85,B 0,C 180,E1 -7619.316,E2 -7619.316} C_VEL
LIN {X 0,Y 471.385,Z 710.867,A -85,B 0,C 180,E1 -7621.836,E2 -7621.836} C_VEL
LIN {X 0,Y 471.904,Z 713.933,A -85,B 0,C 180,E1 -7622.284,E2 -7622.284} C_VEL
LIN {X 0,Y 470.747,Z 737.949,A -85,B 0,C 180,E1 -7625.515,E2 -7625.515} C_VEL
LIN {X 0,Y 469.833,Z 760.486,A -85,B 0,C 180,E1 -7628.5,E2 -7628.5} C_VEL
LIN {X 0,Y 468.878,Z 786.363,A -85,B 0,C 180,E1 -7631.878,E2 -7631.878} C_VEL
LIN {X 0,Y 468.626,Z 794.815,A -85,B 0,C 180,E1 -7632.95,E2 -7632.95} C_VEL
LIN {X 0,Y 471.103,Z 817.606,A -85,B 0,C 180,E1 -7633.41,E2 -7633.41} C_VEL
LIN {X 0,Y 470.434,Z 905.854,A -85,B 0,C 180,E1 -7634.788,E2 -7634.788} C_VEL
LIN {X 0,Y 470.003,Z 919.738,A -85,B 0,C 180,E1 -7635.189,E2 -7635.189} C_VEL
LIN {X 0,Y 469.513,Z 932.745,A -85,B 0,C 180,E1 -7635.755,E2 -7635.755} C_VEL
LIN {X 0,Y 469.023,Z 944.621,A -85,B 0,C 180,E1 -7636.458,E2 -7636.458} C_VEL
LIN {X 0,Y 468.544,Z 955.95,A -85,B 0,C 180,E1 -7637.314,E2 -7637.314} C_VEL
LIN {X 0,Y 468.029,Z 966.48,A -85,B 0,C 180,E1 -7638.303,E2 -7638.303} C_VEL
LIN {X 0,Y 467.651,Z 975.84,A -85,B 0,C 180,E1 -7639.39,E2 -7639.39} C_VEL
LIN {X 0,Y 467.309,Z 984.971,A -85,B 0,C 180,E1 -7640.695,E2 -7640.695} C_VEL
LIN {X 0,Y 467.072,Z 992.34,A -85,B 0,C 180,E1 -7641.998,E2 -7641.998} C_VEL
LIN {X 0,Y 466.933,Z 998.668,A -85,B 0,C 180,E1 -7643.411,E2 -7643.411} C_VEL
LIN {X 0,Y 466.886,Z 1003.534,A -85,B 0,C 180,E1 -7644.817,E2 -7644.817} C_VEL
LIN {X 0,Y 466.878,Z 1005.895,A -85,B 0,C 180,E1 -7645.682,E2 -7645.682} C_VEL
LIN {X 0,Y 466.897,Z 1007.813,A -85,B 0,C 180,E1 -7646.547,E2 -7646.547} C_VEL
LIN {X 0,Y 466.859,Z 1009.246,A -85,B 0,C 180,E1 -7647.41,E2 -7647.41} C_VEL
LIN {X 0,Y 466.846,Z 1010.266,A -85,B 0,C 180,E1 -7648.273,E2 -7648.273} C_VEL
LIN {X 0,Y 466.823,Z 1010.881,A -85,B 0,C 180,E1 -7649.136,E2 -7649.136} C_VEL
LIN {X 0,Y 466.822,Z 1011.096,A -85,B 0,C 180,E1 -7649.999,E2 -7649.999} C_VEL
LIN {X 0,Y 466.825,Z 1010.866,A -85,B 0,C 180,E1 -7650.861,E2 -7650.861} C_VEL
LIN {X 0,Y 466.851,Z 1010.234,A -85,B 0,C 180,E1 -7651.724,E2 -7651.724} C_VEL
LIN {X 0,Y 466.864,Z 1009.197,A -85,B 0,C 180,E1 -7652.587,E2 -7652.587} C_VEL
LIN {X 0,Y 466.896,Z 1007.747,A -85,B 0,C 180,E1 -7653.451,E2 -7653.451} C_VEL
LIN {X 0,Y 466.893,Z 1004.7,A -85,B 0,C 180,E1 -7654.748,E2 -7654.748} C_VEL
LIN {X 0,Y 466.934,Z 999.627,A -85,B 0,C 180,E1 -7656.302,E2 -7656.302} C_VEL
LIN {X 0,Y 467.048,Z 993.229,A -85,B 0,C 180,E1 -7657.782,E2 -7657.782} C_VEL
LIN {X 0,Y 467.258,Z 986.126,A -85,B 0,C 180,E1 -7659.085,E2 -7659.085} C_VEL
LIN {X 0,Y 467.548,Z 977.256,A -85,B 0,C 180,E1 -7660.39,E2 -7660.39} C_VEL
LIN {X 0,Y 467.885,Z 968.188,A -85,B 0,C 180,E1 -7661.479,E2 -7661.479} C_VEL
LIN {X 0,Y 468.424,Z 958.278,A -85,B 0,C 180,E1 -7662.454,E2 -7662.454} C_VEL
LIN {X 0,Y 468.864,Z 947.45,A -85,B 0,C 180,E1 -7663.323,E2 -7663.323} C_VEL
LIN {X 0,Y 469.266,Z 937.335,A -85,B 0,C 180,E1 -7663.973,E2 -7663.973} C_VEL
LIN {X 0,Y 469.783,Z 925.463,A -85,B 0,C 180,E1 -7664.566,E2 -7664.566} C_VEL
LIN {X 0,Y 470.187,Z 912.736,A -85,B 0,C 180,E1 -7665.024,E2 -7665.024} C_VEL
LIN {X 0,Y 470.485,Z 899.788,A -85,B 0,C 180,E1 -7665.319,E2 -7665.319} C_VEL
LIN {X 0,Y 471.009,Z 815.744,A -85,B 0,C 180,E1 -7666.612,E2 -7666.612} C_VEL
LIN {X 0,Y 468.577,Z 793.987,A -85,B 0,C 180,E1 -7667.061,E2 -7667.061} C_VEL
LIN {X 0,Y 469.205,Z 773.823,A -85,B 0,C 180,E1 -7669.648,E2 -7669.648} C_VEL
LIN {X 0,Y 470.105,Z 750.965,A -85,B 0,C 180,E1 -7672.639,E2 -7672.639} C_VEL
LIN {X 0,Y 471.098,Z 726.678,A -85,B 0,C 180,E1 -7675.87,E2 -7675.87} C_VEL
LIN {X 0,Y 471.719,Z 713.047,A -85,B 0,C 180,E1 -7677.713,E2 -7677.713} C_VEL
LIN {X 0,Y 468.158,Z 696.669,A -85,B 0,C 180,E1 -7680.19,E2 -7680.19} C_VEL
LIN {X 0,Y 467.594,Z 694.338,A -85,B 0,C 180,E1 -7680.605,E2 -7680.605} C_VEL
LIN {X 0,Y 467.58,Z 694.236,A -85,B 0,C 180,E1 -7683.787,E2 -7683.787} C_VEL
LIN {X 0,Y 467.541,Z 694.245,A -85,B 0,C 180,E1 -7687.185,E2 -7687.185} C_VEL
LIN {X 0,Y 467.57,Z 694.243,A -85,B 0,C 180,E1 -7690.263,E2 -7690.263} C_VEL
LIN {X 0,Y 467.579,Z 694.242,A -85,B 0,C 180,E1 -7692.566,E2 -7692.566} C_VEL
LIN {X 0,Y 467.563,Z 694.242,A -85,B 0,C 180,E1 -7695.052,E2 -7695.052} C_VEL
LIN {X 0,Y 467.58,Z 694.239,A -85,B 0,C 180,E1 -7697.439,E2 -7697.439} C_VEL
LIN {X 0,Y 467.573,Z 694.238,A -85,B 0,C 180,E1 -7700.854,E2 -7700.854} C_VEL
LIN {X 0,Y 467.553,Z 694.235,A -85,B 0,C 180,E1 -7704.259,E2 -7704.259} C_VEL
LIN {X 0,Y 467.572,Z 694.245,A -85,B 0,C 180,E1 -7707.32,E2 -7707.32} C_VEL
LIN {X 0,Y 467.568,Z 694.24,A -85,B 0,C 180,E1 -7710.665,E2 -7710.665} C_VEL
LIN {X 0,Y 467.617,Z 694.237,A -85,B 0,C 180,E1 -7713.2,E2 -7713.2} C_VEL
LIN {X 0,Y 467.581,Z 694.237,A -85,B 0,C 180,E1 -7716.467,E2 -7716.467} C_VEL
LIN {X 0,Y 467.611,Z 694.24,A -85,B 0,C 180,E1 -7719.777,E2 -7719.777} C_VEL
LIN {X 0,Y 467.597,Z 694.231,A -85,B 0,C 180,E1 -7722.506,E2 -7722.506} C_VEL
LIN {X 0,Y 467.594,Z 694.236,A -85,B 0,C 180,E1 -7725.196,E2 -7725.196} C_VEL
LIN {X 0,Y 467.644,Z 694.233,A -85,B 0,C 180,E1 -7727.854,E2 -7727.854} C_VEL
LIN {X 0,Y 467.669,Z 694.221,A -85,B 0,C 180,E1 -7731.357,E2 -7731.357} C_VEL
LIN {X 0,Y 467.723,Z 694.225,A -85,B 0,C 180,E1 -7733.962,E2 -7733.962} C_VEL
LIN {X 0,Y 467.848,Z 694.203,A -85,B 0,C 180,E1 -7737.417,E2 -7737.417} C_VEL
LIN {X 0,Y 467.869,Z 694.203,A -85,B 0,C 180,E1 -7740,E2 -7740} C_VEL
LIN {X 0,Y 467.847,Z 694.209,A -85,B 0,C 180,E1 -7742.583,E2 -7742.583} C_VEL
LIN {X 0,Y 467.723,Z 694.219,A -85,B 0,C 180,E1 -7746.038,E2 -7746.038} C_VEL
LIN {X 0,Y 467.67,Z 694.229,A -85,B 0,C 180,E1 -7748.643,E2 -7748.643} C_VEL
LIN {X 0,Y 467.645,Z 694.228,A -85,B 0,C 180,E1 -7752.146,E2 -7752.146} C_VEL
LIN {X 0,Y 467.627,Z 694.228,A -85,B 0,C 180,E1 -7755.696,E2 -7755.696} C_VEL
LIN {X 0,Y 467.602,Z 694.239,A -85,B 0,C 180,E1 -7758.764,E2 -7758.764} C_VEL
LIN {X 0,Y 467.569,Z 694.243,A -85,B 0,C 180,E1 -7761.269,E2 -7761.269} C_VEL
LIN {X 0,Y 467.546,Z 694.236,A -85,B 0,C 180,E1 -7763.945,E2 -7763.945} C_VEL
LIN {X 0,Y 467.577,Z 694.241,A -85,B 0,C 180,E1 -7766.803,E2 -7766.803} C_VEL
LIN {X 0,Y 467.543,Z 694.248,A -85,B 0,C 180,E1 -7769.739,E2 -7769.739} C_VEL
LIN {X 0,Y 467.574,Z 694.234,A -85,B 0,C 180,E1 -7772.759,E2 -7772.759} C_VEL
LIN {X 0,Y 467.547,Z 694.243,A -85,B 0,C 180,E1 -7775.891,E2 -7775.891} C_VEL
LIN {X 0,Y 467.574,Z 694.237,A -85,B 0,C 180,E1 -7779.146,E2 -7779.146} C_VEL
LIN {X 0,Y 467.579,Z 694.239,A -85,B 0,C 180,E1 -7782.568,E2 -7782.568} C_VEL
LIN {X 0,Y 467.559,Z 694.243,A -85,B 0,C 180,E1 -7785.054,E2 -7785.054} C_VEL
LIN {X 0,Y 467.573,Z 694.371,A -85,B 0,C 180,E1 -7788.259,E2 -7788.259} C_VEL
LIN {X 0,Y 467.805,Z 695.305,A -85,B 0,C 180,E1 -7788.415,E2 -7788.415} C_VEL
LIN {X 0,Y 471.491,Z 705.299,A -85,B 0,C 180,E1 -7788.734,E2 -7788.734} C_VEL
LIN {X 0,Y 471.016,Z 775.423,A -85,B 0,C 180,E1 -7789.848,E2 -7789.848} C_VEL
LIN {X 0,Y 470.923,Z 788.631,A -85,B 0,C 180,E1 -7790.238,E2 -7790.238} C_VEL
LIN {X 0,Y 470.741,Z 801.666,A -85,B 0,C 180,E1 -7790.812,E2 -7790.812} C_VEL
LIN {X 0,Y 470.511,Z 811.97,A -85,B 0,C 180,E1 -7791.421,E2 -7791.421} C_VEL
LIN {X 0,Y 470.088,Z 822.421,A -85,B 0,C 180,E1 -7792.198,E2 -7792.198} C_VEL
LIN {X 0,Y 469.681,Z 833.487,A -85,B 0,C 180,E1 -7793.237,E2 -7793.237} C_VEL
LIN {X 0,Y 469.205,Z 842.318,A -85,B 0,C 180,E1 -7794.258,E2 -7794.258} C_VEL
LIN {X 0,Y 468.712,Z 851.367,A -85,B 0,C 180,E1 -7795.557,E2 -7795.557} C_VEL
LIN {X 0,Y 468.387,Z 858.243,A -85,B 0,C 180,E1 -7796.788,E2 -7796.788} C_VEL
LIN {X 0,Y 467.992,Z 864.931,A -85,B 0,C 180,E1 -7798.293,E2 -7798.293} C_VEL
LIN {X 0,Y 467.745,Z 869.577,A -85,B 0,C 180,E1 -7799.674,E2 -7799.674} C_VEL
LIN {X 0,Y 467.007,Z 871.572,A -85,B 0,C 180,E1 -7800.35,E2 -7800.35} C_VEL
LIN {X 0,Y 464.026,Z 874.434,A -85,B 0,C 180,E1 -7801.46,E2 -7801.46} C_VEL
LIN {X 0,Y 461.067,Z 876.631,A -85,B 0,C 180,E1 -7802.605,E2 -7802.605} C_VEL
LIN {X 0,Y 460.376,Z 877.402,A -85,B 0,C 180,E1 -7803.329,E2 -7803.329} C_VEL
LIN {X 0,Y 460.32,Z 878.12,A -85,B 0,C 180,E1 -7804.693,E2 -7804.693} C_VEL
LIN {X 0,Y 460.308,Z 877.679,A -85,B 0,C 180,E1 -7806.361,E2 -7806.361} C_VEL
LIN {X 0,Y 460.378,Z 876.451,A -85,B 0,C 180,E1 -7807.566,E2 -7807.566} C_VEL
LIN {X 0,Y 460.499,Z 874.851,A -85,B 0,C 180,E1 -7808.587,E2 -7808.587} C_VEL
LIN {X 0,Y 460.669,Z 871.868,A -85,B 0,C 180,E1 -7809.926,E2 -7809.926} C_VEL
LIN {X 0,Y 460.907,Z 867.606,A -85,B 0,C 180,E1 -7811.326,E2 -7811.326} C_VEL
LIN {X 0,Y 461.248,Z 861.059,A -85,B 0,C 180,E1 -7812.945,E2 -7812.945} C_VEL
LIN {X 0,Y 461.606,Z 853.902,A -85,B 0,C 180,E1 -7814.323,E2 -7814.323} C_VEL
LIN {X 0,Y 462.096,Z 844.873,A -85,B 0,C 180,E1 -7815.693,E2 -7815.693} C_VEL
LIN {X 0,Y 462.522,Z 835.634,A -85,B 0,C 180,E1 -7816.827,E2 -7816.827} C_VEL
LIN {X 0,Y 463.015,Z 825.298,A -85,B 0,C 180,E1 -7817.844,E2 -7817.844} C_VEL
LIN {X 0,Y 463.45,Z 813.828,A -85,B 0,C 180,E1 -7818.742,E2 -7818.742} C_VEL
LIN {X 0,Y 463.779,Z 801.939,A -85,B 0,C 180,E1 -7819.469,E2 -7819.469} C_VEL
LIN {X 0,Y 464.018,Z 789.211,A -85,B 0,C 180,E1 -7820.037,E2 -7820.037} C_VEL
LIN {X 0,Y 464.145,Z 776.018,A -85,B 0,C 180,E1 -7820.435,E2 -7820.435} C_VEL
LIN {X 0,Y 464.457,Z 724.817,A -85,B 0,C 180,E1 -7821.267,E2 -7821.267} C_VEL
LIN {X 0,Y 464.483,Z 706.159,A -85,B 0,C 180,E1 -7821.564,E2 -7821.564} C_VEL
LIN {X 0,Y 460.817,Z 696.079,A -85,B 0,C 180,E1 -7821.886,E2 -7821.886} C_VEL
LIN {X 0,Y 460.649,Z 695.187,A -85,B 0,C 180,E1 -7822.06,E2 -7822.06} C_VEL
LIN {X 0,Y 460.677,Z 695.1,A -85,B 0,C 180,E1 -7824.749,E2 -7824.749} C_VEL
LIN {X 0,Y 460.758,Z 695.09,A -85,B 0,C 180,E1 -7827.379,E2 -7827.379} C_VEL
LIN {X 0,Y 460.822,Z 695.083,A -85,B 0,C 180,E1 -7830.001,E2 -7830.001} C_VEL
LIN {X 0,Y 460.757,Z 695.093,A -85,B 0,C 180,E1 -7832.624,E2 -7832.624} C_VEL
LIN {X 0,Y 460.671,Z 695.104,A -85,B 0,C 180,E1 -7836.132,E2 -7836.132} C_VEL
LIN {X 0,Y 460.589,Z 695.113,A -85,B 0,C 180,E1 -7838.778,E2 -7838.778} C_VEL
LIN {X 0,Y 460.603,Z 695.111,A -85,B 0,C 180,E1 -7842.436,E2 -7842.436} C_VEL
LIN {X 0,Y 460.585,Z 695.106,A -85,B 0,C 180,E1 -7845.989,E2 -7845.989} C_VEL
LIN {X 0,Y 460.541,Z 695.114,A -85,B 0,C 180,E1 -7848.889,E2 -7848.889} C_VEL
LIN {X 0,Y 460.519,Z 695.117,A -85,B 0,C 180,E1 -7851.487,E2 -7851.487} C_VEL
LIN {X 0,Y 460.517,Z 695.117,A -85,B 0,C 180,E1 -7854.335,E2 -7854.335} C_VEL
LIN {X 0,Y 460.49,Z 695.118,A -85,B 0,C 180,E1 -7857.25,E2 -7857.25} C_VEL
LIN {X 0,Y 460.484,Z 695.121,A -85,B 0,C 180,E1 -7860.243,E2 -7860.243} C_VEL
LIN {X 0,Y 460.504,Z 695.114,A -85,B 0,C 180,E1 -7863.328,E2 -7863.328} C_VEL
LIN {X 0,Y 460.46,Z 695.115,A -85,B 0,C 180,E1 -7866.532,E2 -7866.532} C_VEL
LIN {X 0,Y 460.48,Z 695.124,A -85,B 0,C 180,E1 -7869.869,E2 -7869.869} C_VEL
LIN {X 0,Y 460.462,Z 695.124,A -85,B 0,C 180,E1 -7872.893,E2 -7872.893} C_VEL
LIN {X 0,Y 460.509,Z 695.124,A -85,B 0,C 180,E1 -7875.832,E2 -7875.832} C_VEL
LIN {X 0,Y 460.509,Z 695.118,A -85,B 0,C 180,E1 -7878.986,E2 -7878.986} C_VEL
LIN {X 0,Y 460.482,Z 695.124,A -85,B 0,C 180,E1 -7882.375,E2 -7882.375} C_VEL
LIN {X 0,Y 460.519,Z 695.122,A -85,B 0,C 180,E1 -7885.621,E2 -7885.621} C_VEL
LIN {X 0,Y 460.511,Z 695.123,A -85,B 0,C 180,E1 -7888.742,E2 -7888.742} C_VEL
LIN {X 0,Y 460.532,Z 695.385,A -85,B 0,C 180,E1 -7890.263,E2 -7890.263} C_VEL
LIN {X 0,Y 460.783,Z 696.435,A -85,B 0,C 180,E1 -7890.389,E2 -7890.389} C_VEL
LIN {X 0,Y 464.178,Z 705.898,A -85,B 0,C 180,E1 -7890.684,E2 -7890.684} C_VEL
LIN {X 0,Y 463.587,Z 771.481,A -85,B 0,C 180,E1 -7891.793,E2 -7891.793} C_VEL
LIN {X 0,Y 463.47,Z 782.628,A -85,B 0,C 180,E1 -7892.114,E2 -7892.114} C_VEL
LIN {X 0,Y 463.218,Z 793.526,A -85,B 0,C 180,E1 -7892.558,E2 -7892.558} C_VEL
LIN {X 0,Y 463.027,Z 802.463,A -85,B 0,C 180,E1 -7893.025,E2 -7893.025} C_VEL
LIN {X 0,Y 462.703,Z 812.202,A -85,B 0,C 180,E1 -7893.659,E2 -7893.659} C_VEL
LIN {X 0,Y 462.341,Z 822.003,A -85,B 0,C 180,E1 -7894.448,E2 -7894.448} C_VEL
LIN {X 0,Y 461.928,Z 830.464,A -85,B 0,C 180,E1 -7895.266,E2 -7895.266} C_VEL
LIN {X 0,Y 461.643,Z 837.795,A -85,B 0,C 180,E1 -7896.103,E2 -7896.103} C_VEL
LIN {X 0,Y 461.316,Z 845.397,A -85,B 0,C 180,E1 -7897.139,E2 -7897.139} C_VEL
LIN {X 0,Y 461.04,Z 851.488,A -85,B 0,C 180,E1 -7898.117,E2 -7898.117} C_VEL
LIN {X 0,Y 460.677,Z 858.277,A -85,B 0,C 180,E1 -7899.458,E2 -7899.458} C_VEL
LIN {X 0,Y 460.535,Z 862.218,A -85,B 0,C 180,E1 -7900.383,E2 -7900.383} C_VEL
LIN {X 0,Y 460.363,Z 866.9,A -85,B 0,C 180,E1 -7901.762,E2 -7901.762} C_VEL
LIN {X 0,Y 460.189,Z 870.376,A -85,B 0,C 180,E1 -7903.132,E2 -7903.132} C_VEL
LIN {X 0,Y 460.132,Z 872.381,A -85,B 0,C 180,E1 -7904.211,E2 -7904.211} C_VEL
LIN {X 0,Y 460.045,Z 874.212,A -85,B 0,C 180,E1 -7905.852,E2 -7905.852} C_VEL
LIN {X 0,Y 460.051,Z 874.615,A -85,B 0,C 180,E1 -7906.753,E2 -7906.753} C_VEL
LIN {X 0,Y 460.104,Z 874.548,A -85,B 0,C 180,E1 -7907.851,E2 -7907.851} C_VEL
LIN {X 0,Y 460.188,Z 873.279,A -85,B 0,C 180,E1 -7909.44,E2 -7909.44} C_VEL
LIN {X 0,Y 460.31,Z 870.352,A -85,B 0,C 180,E1 -7911.218,E2 -7911.218} C_VEL
LIN {X 0,Y 460.535,Z 866.352,A -85,B 0,C 180,E1 -7912.724,E2 -7912.724} C_VEL
LIN {X 0,Y 460.71,Z 862.414,A -85,B 0,C 180,E1 -7913.87,E2 -7913.87} C_VEL
LIN {X 0,Y 460.917,Z 856.659,A -85,B 0,C 180,E1 -7915.189,E2 -7915.189} C_VEL
LIN {X 0,Y 461.23,Z 850.778,A -85,B 0,C 180,E1 -7916.287,E2 -7916.287} C_VEL
LIN {X 0,Y 461.607,Z 843.682,A -85,B 0,C 180,E1 -7917.382,E2 -7917.382} C_VEL
LIN {X 0,Y 461.909,Z 837.017,A -85,B 0,C 180,E1 -7918.256,E2 -7918.256} C_VEL
LIN {X 0,Y 462.304,Z 827.968,A -85,B 0,C 180,E1 -7919.238,E2 -7919.238} C_VEL
LIN {X 0,Y 462.675,Z 819.518,A -85,B 0,C 180,E1 -7920,E2 -7920} C_VEL
LIN {X 0,Y 462.995,Z 810.862,A -85,B 0,C 180,E1 -7920.652,E2 -7920.652} C_VEL
LIN {X 0,Y 463.268,Z 800.037,A -85,B 0,C 180,E1 -7921.304,E2 -7921.304} C_VEL
LIN {X 0,Y 463.539,Z 789.485,A -85,B 0,C 180,E1 -7921.792,E2 -7921.792} C_VEL
LIN {X 0,Y 463.626,Z 779.329,A -85,B 0,C 180,E1 -7922.145,E2 -7922.145} C_VEL
LIN {X 0,Y 463.68,Z 766.164,A -85,B 0,C 180,E1 -7922.443,E2 -7922.443} C_VEL
LIN {X 0,Y 464.333,Z 705.372,A -85,B 0,C 180,E1 -7923.471,E2 -7923.471} C_VEL
LIN {X 0,Y 460.776,Z 696.171,A -85,B 0,C 180,E1 -7923.799,E2 -7923.799} C_VEL
LIN {X 0,Y 460.589,Z 695.222,A -85,B 0,C 180,E1 -7923.965,E2 -7923.965} C_VEL
LIN {X 0,Y 460.691,Z 695.102,A -85,B 0,C 180,E1 -7926.13,E2 -7926.13} C_VEL
LIN {X 0,Y 460.626,Z 695.108,A -85,B 0,C 180,E1 -7928.776,E2 -7928.776} C_VEL
LIN {X 0,Y 460.621,Z 695.111,A -85,B 0,C 180,E1 -7932.445,E2 -7932.445} C_VEL
LIN {X 0,Y 460.608,Z 695.111,A -85,B 0,C 180,E1 -7935.997,E2 -7935.997} C_VEL
LIN {X 0,Y 460.575,Z 695.111,A -85,B 0,C 180,E1 -7939.615,E2 -7939.615} C_VEL
LIN {X 0,Y 460.518,Z 695.123,A -85,B 0,C 180,E1 -7942.428,E2 -7942.428} C_VEL
LIN {X 0,Y 460.555,Z 695.113,A -85,B 0,C 180,E1 -7945.796,E2 -7945.796} C_VEL
LIN {X 0,Y 460.533,Z 695.118,A -85,B 0,C 180,E1 -7948.234,E2 -7948.234} C_VEL
LIN {X 0,Y 460.527,Z 695.12,A -85,B 0,C 180,E1 -7951.282,E2 -7951.282} C_VEL
LIN {X 0,Y 460.529,Z 695.118,A -85,B 0,C 180,E1 -7954.503,E2 -7954.503} C_VEL
LIN {X 0,Y 460.507,Z 695.121,A -85,B 0,C 180,E1 -7957.623,E2 -7957.623} C_VEL
LIN {X 0,Y 460.548,Z 695.114,A -85,B 0,C 180,E1 -7960.269,E2 -7960.269} C_VEL
LIN {X 0,Y 460.505,Z 695.124,A -85,B 0,C 180,E1 -7963.375,E2 -7963.375} C_VEL
LIN {X 0,Y 460.503,Z 695.12,A -85,B 0,C 180,E1 -7966.624,E2 -7966.624} C_VEL
LIN {X 0,Y 460.544,Z 695.119,A -85,B 0,C 180,E1 -7969.73,E2 -7969.73} C_VEL
LIN {X 0,Y 460.502,Z 695.119,A -85,B 0,C 180,E1 -7972.524,E2 -7972.524} C_VEL
LIN {X 0,Y 460.542,Z 695.12,A -85,B 0,C 180,E1 -7975.622,E2 -7975.622} C_VEL
LIN {X 0,Y 460.556,Z 695.231,A -85,B 0,C 180,E1 -7979.016,E2 -7979.016} C_VEL
LIN {X 0,Y 463.742,Z 709.008,A -85,B 0,C 180,E1 -7981.205,E2 -7981.205} C_VEL
LIN {X 0,Y 464.928,Z 714.622,A -85,B 0,C 180,E1 -7982.055,E2 -7982.055} C_VEL
LIN {X 0,Y 464.119,Z 733.66,A -85,B 0,C 180,E1 -7984.672,E2 -7984.672} C_VEL
LIN {X 0,Y 462.904,Z 759.78,A -85,B 0,C 180,E1 -7988.192,E2 -7988.192} C_VEL
LIN {X 0,Y 461.848,Z 787.096,A -85,B 0,C 180,E1 -7991.822,E2 -7991.822} C_VEL
LIN {X 0,Y 461.637,Z 793.618,A -85,B 0,C 180,E1 -7992.672,E2 -7992.672} C_VEL
LIN {X 0,Y 464.268,Z 818.526,A -85,B 0,C 180,E1 -7993.19,E2 -7993.19} C_VEL
LIN {X 0,Y 463.568,Z 904.757,A -85,B 0,C 180,E1 -7994.557,E2 -7994.557} C_VEL
LIN {X 0,Y 463.125,Z 918.68,A -85,B 0,C 180,E1 -7994.964,E2 -7994.964} C_VEL
LIN {X 0,Y 462.607,Z 931.712,A -85,B 0,C 180,E1 -7995.538,E2 -7995.538} C_VEL
LIN {X 0,Y 462.043,Z 943.591,A -85,B 0,C 180,E1 -7996.25,E2 -7996.25} C_VEL
LIN {X 0,Y 461.518,Z 954.217,A -85,B 0,C 180,E1 -7997.057,E2 -7997.057} C_VEL
LIN {X 0,Y 461.115,Z 964.398,A -85,B 0,C 180,E1 -7998.013,E2 -7998.013} C_VEL
LIN {X 0,Y 460.682,Z 973.099,A -85,B 0,C 180,E1 -7999.005,E2 -7999.005} C_VEL
LIN {X 0,Y 460.344,Z 981.15,A -85,B 0,C 180,E1 -8000.109,E2 -8000.109} C_VEL
LIN {X 0,Y 460.097,Z 989.044,A -85,B 0,C 180,E1 -8001.434,E2 -8001.434} C_VEL
LIN {X 0,Y 459.92,Z 996.321,A -85,B 0,C 180,E1 -8002.977,E2 -8002.977} C_VEL
LIN {X 0,Y 459.868,Z 1001.178,A -85,B 0,C 180,E1 -8004.298,E2 -8004.298} C_VEL
LIN {X 0,Y 459.833,Z 1004.891,A -85,B 0,C 180,E1 -8005.616,E2 -8005.616} C_VEL
LIN {X 0,Y 459.855,Z 1006.81,A -85,B 0,C 180,E1 -8006.494,E2 -8006.494} C_VEL
LIN {X 0,Y 459.818,Z 1008.243,A -85,B 0,C 180,E1 -8007.371,E2 -8007.371} C_VEL
LIN {X 0,Y 459.811,Z 1009.261,A -85,B 0,C 180,E1 -8008.247,E2 -8008.247} C_VEL
LIN {X 0,Y 459.793,Z 1009.876,A -85,B 0,C 180,E1 -8009.123,E2 -8009.123} C_VEL
LIN {X 0,Y 459.794,Z 1010.09,A -85,B 0,C 180,E1 -8009.999,E2 -8009.999} C_VEL
LIN {X 0,Y 459.795,Z 1009.858,A -85,B 0,C 180,E1 -8010.874,E2 -8010.874} C_VEL
LIN {X 0,Y 459.816,Z 1009.222,A -85,B 0,C 180,E1 -8011.75,E2 -8011.75} C_VEL
LIN {X 0,Y 459.825,Z 1008.181,A -85,B 0,C 180,E1 -8012.627,E2 -8012.627} C_VEL
LIN {X 0,Y 459.854,Z 1006.729,A -85,B 0,C 180,E1 -8013.503,E2 -8013.503} C_VEL
LIN {X 0,Y 459.852,Z 1003.675,A -85,B 0,C 180,E1 -8014.82,E2 -8014.82} C_VEL
LIN {X 0,Y 459.901,Z 999.556,A -85,B 0,C 180,E1 -8016.139,E2 -8016.139} C_VEL
LIN {X 0,Y 459.976,Z 993.23,A -85,B 0,C 180,E1 -8017.682,E2 -8017.682} C_VEL
LIN {X 0,Y 460.145,Z 986.343,A -85,B 0,C 180,E1 -8019.005,E2 -8019.005} C_VEL
LIN {X 0,Y 460.457,Z 977.831,A -85,B 0,C 180,E1 -8020.33,E2 -8020.33} C_VEL
LIN {X 0,Y 460.807,Z 968.117,A -85,B 0,C 180,E1 -8021.546,E2 -8021.546} C_VEL
LIN {X 0,Y 461.402,Z 957.792,A -85,B 0,C 180,E1 -8022.593,E2 -8022.593} C_VEL
LIN {X 0,Y 461.898,Z 946.38,A -85,B 0,C 180,E1 -8023.528,E2 -8023.528} C_VEL
LIN {X 0,Y 462.427,Z 934.296,A -85,B 0,C 180,E1 -8024.297,E2 -8024.297} C_VEL
LIN {X 0,Y 462.963,Z 921.771,A -85,B 0,C 180,E1 -8024.898,E2 -8024.898} C_VEL
LIN {X 0,Y 463.451,Z 908.904,A -85,B 0,C 180,E1 -8025.332,E2 -8025.332} C_VEL
LIN {X 0,Y 463.673,Z 895.328,A -85,B 0,C 180,E1 -8025.606,E2 -8025.606} C_VEL
LIN {X 0,Y 464.136,Z 816.124,A -85,B 0,C 180,E1 -8026.844,E2 -8026.844} C_VEL
LIN {X 0,Y 461.564,Z 792.944,A -85,B 0,C 180,E1 -8027.329,E2 -8027.329} C_VEL
LIN {X 0,Y 462.186,Z 774.172,A -85,B 0,C 180,E1 -8029.774,E2 -8029.774} C_VEL
LIN {X 0,Y 463.223,Z 749.979,A -85,B 0,C 180,E1 -8032.995,E2 -8032.995} C_VEL
LIN {X 0,Y 464.33,Z 724.645,A -85,B 0,C 180,E1 -8036.431,E2 -8036.431} C_VEL
LIN {X 0,Y 464.723,Z 713.628,A -85,B 0,C 180,E1 -8037.956,E2 -8037.956} C_VEL
LIN {X 0,Y 461.066,Z 697.51,A -85,B 0,C 180,E1 -8040.451,E2 -8040.451} C_VEL
LIN {X 0,Y 460.543,Z 695.212,A -85,B 0,C 180,E1 -8040.87,E2 -8040.87} C_VEL
LIN {X 0,Y 460.54,Z 695.113,A -85,B 0,C 180,E1 -8044.375,E2 -8044.375} C_VEL
LIN {X 0,Y 460.494,Z 695.122,A -85,B 0,C 180,E1 -8047.622,E2 -8047.622} C_VEL
LIN {X 0,Y 460.534,Z 695.119,A -85,B 0,C 180,E1 -8050.268,E2 -8050.268} C_VEL
LIN {X 0,Y 460.492,Z 695.12,A -85,B 0,C 180,E1 -8053.374,E2 -8053.374} C_VEL
LIN {X 0,Y 460.505,Z 695.119,A -85,B 0,C 180,E1 -8056.625,E2 -8056.625} C_VEL
LIN {X 0,Y 460.534,Z 695.109,A -85,B 0,C 180,E1 -8059.729,E2 -8059.729} C_VEL
LIN {X 0,Y 460.518,Z 695.119,A -85,B 0,C 180,E1 -8062.518,E2 -8062.518} C_VEL
LIN {X 0,Y 460.539,Z 695.115,A -85,B 0,C 180,E1 -8065.623,E2 -8065.623} C_VEL
LIN {X 0,Y 460.526,Z 695.118,A -85,B 0,C 180,E1 -8068.744,E2 -8068.744} C_VEL
LIN {X 0,Y 460.548,Z 695.115,A -85,B 0,C 180,E1 -8071.767,E2 -8071.767} C_VEL
LIN {X 0,Y 460.548,Z 695.112,A -85,B 0,C 180,E1 -8074.705,E2 -8074.705} C_VEL
LIN {X 0,Y 460.5,Z 695.124,A -85,B 0,C 180,E1 -8077.571,E2 -8077.571} C_VEL
LIN {X 0,Y 460.557,Z 695.112,A -85,B 0,C 180,E1 -8080.384,E2 -8080.384} C_VEL
LIN {X 0,Y 460.619,Z 695.109,A -85,B 0,C 180,E1 -8084.06,E2 -8084.06} C_VEL
LIN {X 0,Y 460.597,Z 695.108,A -85,B 0,C 180,E1 -8087.666,E2 -8087.666} C_VEL
LIN {X 0,Y 460.616,Z 695.099,A -85,B 0,C 180,E1 -8091.224,E2 -8091.224} C_VEL
LIN {X 0,Y 460.689,Z 695.1,A -85,B 0,C 180,E1 -8093.87,E2 -8093.87} C_VEL
LIN {X 0,Y 460.813,Z 695.079,A -85,B 0,C 180,E1 -8097.378,E2 -8097.378} C_VEL
LIN {X 0,Y 460.84,Z 695.078,A -85,B 0,C 180,E1 -8100,E2 -8100} C_VEL
LIN {X 0,Y 460.812,Z 695.085,A -85,B 0,C 180,E1 -8102.623,E2 -8102.623} C_VEL
LIN {X 0,Y 460.69,Z 695.097,A -85,B 0,C 180,E1 -8106.13,E2 -8106.13} C_VEL
LIN {X 0,Y 460.617,Z 695.107,A -85,B 0,C 180,E1 -8108.777,E2 -8108.777} C_VEL
LIN {X 0,Y 460.601,Z 695.109,A -85,B 0,C 180,E1 -8112.445,E2 -8112.445} C_VEL
LIN {X 0,Y 460.588,Z 695.104,A -85,B 0,C 180,E1 -8115.998,E2 -8115.998} C_VEL
LIN {X 0,Y 460.557,Z 695.113,A -85,B 0,C 180,E1 -8119.616,E2 -8119.616} C_VEL
LIN {X 0,Y 460.499,Z 695.117,A -85,B 0,C 180,E1 -8122.43,E2 -8122.43} C_VEL
LIN {X 0,Y 460.535,Z 695.118,A -85,B 0,C 180,E1 -8125.797,E2 -8125.797} C_VEL
LIN {X 0,Y 460.539,Z 695.108,A -85,B 0,C 180,E1 -8128.234,E2 -8128.234} C_VEL
LIN {X 0,Y 460.512,Z 695.126,A -85,B 0,C 180,E1 -8131.284,E2 -8131.284} C_VEL
LIN {X 0,Y 460.524,Z 695.117,A -85,B 0,C 180,E1 -8134.507,E2 -8134.507} C_VEL
LIN {X 0,Y 460.52,Z 695.125,A -85,B 0,C 180,E1 -8137.622,E2 -8137.622} C_VEL
LIN {X 0,Y 460.534,Z 695.118,A -85,B 0,C 180,E1 -8140.271,E2 -8140.271} C_VEL
LIN {X 0,Y 460.491,Z 695.122,A -85,B 0,C 180,E1 -8143.377,E2 -8143.377} C_VEL
LIN {X 0,Y 460.502,Z 695.116,A -85,B 0,C 180,E1 -8146.627,E2 -8146.627} C_VEL
LIN {X 0,Y 460.542,Z 695.294,A -85,B 0,C 180,E1 -8148.005,E2 -8148.005} C_VEL
LIN {X 0,Y 460.804,Z 696.37,A -85,B 0,C 180,E1 -8148.155,E2 -8148.155} C_VEL
LIN {X 0,Y 464.637,Z 706.612,A -85,B 0,C 180,E1 -8148.489,E2 -8148.489} C_VEL
LIN {X 0,Y 464.214,Z 776.383,A -85,B 0,C 180,E1 -8149.617,E2 -8149.617} C_VEL
LIN {X 0,Y 464.131,Z 789.699,A -85,B 0,C 180,E1 -8150.016,E2 -8150.016} C_VEL
LIN {X 0,Y 463.939,Z 802.489,A -85,B 0,C 180,E1 -8150.586,E2 -8150.586} C_VEL
LIN {X 0,Y 463.646,Z 814.206,A -85,B 0,C 180,E1 -8151.3,E2 -8151.3} C_VEL
LIN {X 0,Y 463.196,Z 824.473,A -85,B 0,C 180,E1 -8152.092,E2 -8152.092} C_VEL
LIN {X 0,Y 462.789,Z 835.325,A -85,B 0,C 180,E1 -8153.143,E2 -8153.143} C_VEL
LIN {X 0,Y 462.3,Z 844.007,A -85,B 0,C 180,E1 -8154.179,E2 -8154.179} C_VEL
LIN {X 0,Y 461.775,Z 852.874,A -85,B 0,C 180,E1 -8155.493,E2 -8155.493} C_VEL
LIN {X 0,Y 461.371,Z 860.496,A -85,B 0,C 180,E1 -8156.91,E2 -8156.91} C_VEL
LIN {X 0,Y 461.014,Z 866.181,A -85,B 0,C 180,E1 -8158.247,E2 -8158.247} C_VEL
LIN {X 0,Y 460.751,Z 871.138,A -85,B 0,C 180,E1 -8159.779,E2 -8159.779} C_VEL
LIN {X 0,Y 460.612,Z 873.626,A -85,B 0,C 180,E1 -8160.776,E2 -8160.776} C_VEL
LIN {X 0,Y 460.454,Z 876.32,A -85,B 0,C 180,E1 -8162.285,E2 -8162.285} C_VEL
LIN {X 0,Y 460.376,Z 877.402,A -85,B 0,C 180,E1 -8163.329,E2 -8163.329} C_VEL
LIN {X 0,Y 459.695,Z 878.035,A -85,B 0,C 180,E1 -8164.055,E2 -8164.055} C_VEL
LIN {X 0,Y 456.797,Z 878.636,A -85,B 0,C 180,E1 -8165.238,E2 -8165.238} C_VEL
LIN {X 0,Y 454.379,Z 878.631,A -85,B 0,C 180,E1 -8166.192,E2 -8166.192} C_VEL
LIN {X 0,Y 453.378,Z 878.207,A -85,B 0,C 180,E1 -8166.928,E2 -8166.928} C_VEL
LIN {X 0,Y 453.317,Z 877.981,A -85,B 0,C 180,E1 -8167.177,E2 -8167.177} C_VEL
LIN {X 0,Y 453.462,Z 876.22,A -85,B 0,C 180,E1 -8168.422,E2 -8168.422} C_VEL
LIN {X 0,Y 453.683,Z 872.652,A -85,B 0,C 180,E1 -8170.076,E2 -8170.076} C_VEL
LIN {X 0,Y 453.935,Z 868.324,A -85,B 0,C 180,E1 -8171.496,E2 -8171.496} C_VEL
LIN {X 0,Y 454.238,Z 862.75,A -85,B 0,C 180,E1 -8172.906,E2 -8172.906} C_VEL
LIN {X 0,Y 454.622,Z 855.757,A -85,B 0,C 180,E1 -8174.306,E2 -8174.306} C_VEL
LIN {X 0,Y 455.065,Z 848.575,A -85,B 0,C 180,E1 -8175.467,E2 -8175.467} C_VEL
LIN {X 0,Y 455.525,Z 839.89,A -85,B 0,C 180,E1 -8176.62,E2 -8176.62} C_VEL
LIN {X 0,Y 455.973,Z 830.341,A -85,B 0,C 180,E1 -8177.653,E2 -8177.653} C_VEL
LIN {X 0,Y 456.424,Z 819.91,A -85,B 0,C 180,E1 -8178.567,E2 -8178.567} C_VEL
LIN {X 0,Y 456.847,Z 808.47,A -85,B 0,C 180,E1 -8179.363,E2 -8179.363} C_VEL
LIN {X 0,Y 457.097,Z 796.981,A -85,B 0,C 180,E1 -8179.977,E2 -8179.977} C_VEL
LIN {X 0,Y 457.279,Z 783.569,A -85,B 0,C 180,E1 -8180.487,E2 -8180.487} C_VEL
LIN {X 0,Y 457.329,Z 769.982,A -85,B 0,C 180,E1 -8180.805,E2 -8180.805} C_VEL
LIN {X 0,Y 457.684,Z 707.652,A -85,B 0,C 180,E1 -8181.803,E2 -8181.803} C_VEL
LIN {X 0,Y 453.761,Z 696.817,A -85,B 0,C 180,E1 -8182.162,E2 -8182.162} C_VEL
LIN {X 0,Y 453.618,Z 696.067,A -85,B 0,C 180,E1 -8182.322,E2 -8182.322} C_VEL
LIN {X 0,Y 453.65,Z 695.977,A -85,B 0,C 180,E1 -8184.668,E2 -8184.668} C_VEL
LIN {X 0,Y 453.69,Z 695.973,A -85,B 0,C 180,E1 -8188.226,E2 -8188.226} C_VEL
LIN {X 0,Y 453.771,Z 695.962,A -85,B 0,C 180,E1 -8190.001,E2 -8190.001} C_VEL
LIN {X 0,Y 453.704,Z 695.972,A -85,B 0,C 180,E1 -8192.665,E2 -8192.665} C_VEL
LIN {X 0,Y 453.639,Z 695.981,A -85,B 0,C 180,E1 -8196.227,E2 -8196.227} C_VEL
LIN {X 0,Y 453.559,Z 695.987,A -85,B 0,C 180,E1 -8198.915,E2 -8198.915} C_VEL
LIN {X 0,Y 453.57,Z 695.988,A -85,B 0,C 180,E1 -8202.53,E2 -8202.53} C_VEL
LIN {X 0,Y 453.543,Z 695.984,A -85,B 0,C 180,E1 -8206.197,E2 -8206.197} C_VEL
LIN {X 0,Y 453.492,Z 695.99,A -85,B 0,C 180,E1 -8209.028,E2 -8209.028} C_VEL
LIN {X 0,Y 453.48,Z 695.992,A -85,B 0,C 180,E1 -8211.837,E2 -8211.837} C_VEL
LIN {X 0,Y 453.466,Z 695.999,A -85,B 0,C 180,E1 -8214.738,E2 -8214.738} C_VEL
LIN {X 0,Y 453.462,Z 695.991,A -85,B 0,C 180,E1 -8217.942,E2 -8217.942} C_VEL
LIN {X 0,Y 453.453,Z 696,A -85,B 0,C 180,E1 -8220.763,E2 -8220.763} C_VEL
LIN {X 0,Y 453.458,Z 695.984,A -85,B 0,C 180,E1 -8223.916,E2 -8223.916} C_VEL
LIN {X 0,Y 453.437,Z 695.995,A -85,B 0,C 180,E1 -8227.192,E2 -8227.192} C_VEL
LIN {X 0,Y 453.47,Z 695.994,A -85,B 0,C 180,E1 -8230.613,E2 -8230.613} C_VEL
LIN {X 0,Y 453.447,Z 695.999,A -85,B 0,C 180,E1 -8234.225,E2 -8234.225} C_VEL
LIN {X 0,Y 453.421,Z 696.001,A -85,B 0,C 180,E1 -8237,E2 -8237} C_VEL
LIN {X 0,Y 453.473,Z 695.998,A -85,B 0,C 180,E1 -8239.414,E2 -8239.414} C_VEL
LIN {X 0,Y 453.433,Z 696,A -85,B 0,C 180,E1 -8242.808,E2 -8242.808} C_VEL
LIN {X 0,Y 453.454,Z 696.003,A -85,B 0,C 180,E1 -8246.085,E2 -8246.085} C_VEL
LIN {X 0,Y 453.456,Z 696.003,A -85,B 0,C 180,E1 -8249.239,E2 -8249.239} C_VEL
LIN {X 0,Y 453.503,Z 696.27,A -85,B 0,C 180,E1 -8250.023,E2 -8250.023} C_VEL
LIN {X 0,Y 453.769,Z 697.432,A -85,B 0,C 180,E1 -8250.152,E2 -8250.152} C_VEL
LIN {X 0,Y 457.421,Z 707.511,A -85,B 0,C 180,E1 -8250.468,E2 -8250.468} C_VEL
LIN {X 0,Y 456.744,Z 771.928,A -85,B 0,C 180,E1 -8251.573,E2 -8251.573} C_VEL
LIN {X 0,Y 456.597,Z 783.467,A -85,B 0,C 180,E1 -8251.907,E2 -8251.907} C_VEL
LIN {X 0,Y 456.343,Z 794.393,A -85,B 0,C 180,E1 -8252.358,E2 -8252.358} C_VEL
LIN {X 0,Y 456.146,Z 804.068,A -85,B 0,C 180,E1 -8252.879,E2 -8252.879} C_VEL
LIN {X 0,Y 455.796,Z 813.91,A -85,B 0,C 180,E1 -8253.539,E2 -8253.539} C_VEL
LIN {X 0,Y 455.44,Z 822.927,A -85,B 0,C 180,E1 -8254.278,E2 -8254.278} C_VEL
LIN {X 0,Y 455.019,Z 831.404,A -85,B 0,C 180,E1 -8255.109,E2 -8255.109} C_VEL
LIN {X 0,Y 454.695,Z 839.235,A -85,B 0,C 180,E1 -8256.025,E2 -8256.025} C_VEL
LIN {X 0,Y 454.37,Z 846.363,A -85,B 0,C 180,E1 -8257.011,E2 -8257.011} C_VEL
LIN {X 0,Y 453.968,Z 853.816,A -85,B 0,C 180,E1 -8258.263,E2 -8258.263} C_VEL
LIN {X 0,Y 453.747,Z 858.266,A -85,B 0,C 180,E1 -8259.13,E2 -8259.13} C_VEL
LIN {X 0,Y 453.518,Z 864.204,A -85,B 0,C 180,E1 -8260.585,E2 -8260.585} C_VEL
LIN {X 0,Y 453.305,Z 868.512,A -85,B 0,C 180,E1 -8261.936,E2 -8261.936} C_VEL
LIN {X 0,Y 453.201,Z 870.917,A -85,B 0,C 180,E1 -8262.864,E2 -8262.864} C_VEL
LIN {X 0,Y 453.109,Z 873.225,A -85,B 0,C 180,E1 -8264.086,E2 -8264.086} C_VEL
LIN {X 0,Y 453.047,Z 875.096,A -85,B 0,C 180,E1 -8265.629,E2 -8265.629} C_VEL
LIN {X 0,Y 453.049,Z 875.588,A -85,B 0,C 180,E1 -8266.544,E2 -8266.544} C_VEL
LIN {X 0,Y 453.094,Z 875.637,A -85,B 0,C 180,E1 -8267.746,E2 -8267.746} C_VEL
LIN {X 0,Y 453.157,Z 874.526,A -85,B 0,C 180,E1 -8269.274,E2 -8269.274} C_VEL
LIN {X 0,Y 453.314,Z 871.843,A -85,B 0,C 180,E1 -8271.081,E2 -8271.081} C_VEL
LIN {X 0,Y 453.56,Z 867.2,A -85,B 0,C 180,E1 -8272.879,E2 -8272.879} C_VEL
LIN {X 0,Y 453.73,Z 864.277,A -85,B 0,C 180,E1 -8273.775,E2 -8273.775} C_VEL
LIN {X 0,Y 453.977,Z 857.62,A -85,B 0,C 180,E1 -8275.338,E2 -8275.338} C_VEL
LIN {X 0,Y 454.319,Z 851.72,A -85,B 0,C 180,E1 -8276.452,E2 -8276.452} C_VEL
LIN {X 0,Y 454.725,Z 844.601,A -85,B 0,C 180,E1 -8277.564,E2 -8277.564} C_VEL
LIN {X 0,Y 455.048,Z 837.891,A -85,B 0,C 180,E1 -8278.451,E2 -8278.451} C_VEL
LIN {X 0,Y 455.466,Z 828.787,A -85,B 0,C 180,E1 -8279.447,E2 -8279.447} C_VEL
LIN {X 0,Y 455.853,Z 820.268,A -85,B 0,C 180,E1 -8280.221,E2 -8280.221} C_VEL
LIN {X 0,Y 456.183,Z 811.521,A -85,B 0,C 180,E1 -8280.883,E2 -8280.883} C_VEL
LIN {X 0,Y 456.44,Z 801.656,A -85,B 0,C 180,E1 -8281.489,E2 -8281.489} C_VEL
LIN {X 0,Y 456.741,Z 790.535,A -85,B 0,C 180,E1 -8282.011,E2 -8282.011} C_VEL
LIN {X 0,Y 456.827,Z 780.356,A -85,B 0,C 180,E1 -8282.369,E2 -8282.369} C_VEL
LIN {X 0,Y 456.89,Z 768.782,A -85,B 0,C 180,E1 -8282.645,E2 -8282.645} C_VEL
LIN {X 0,Y 457.615,Z 707.064,A -85,B 0,C 180,E1 -8283.714,E2 -8283.714} C_VEL
LIN {X 0,Y 453.712,Z 696.919,A -85,B 0,C 180,E1 -8284.098,E2 -8284.098} C_VEL
LIN {X 0,Y 453.523,Z 696.068,A -85,B 0,C 180,E1 -8284.281,E2 -8284.281} C_VEL
LIN {X 0,Y 453.657,Z 695.978,A -85,B 0,C 180,E1 -8286.225,E2 -8286.225} C_VEL
LIN {X 0,Y 453.592,Z 695.984,A -85,B 0,C 180,E1 -8288.913,E2 -8288.913} C_VEL
LIN {X 0,Y 453.571,Z 695.988,A -85,B 0,C 180,E1 -8292.529,E2 -8292.529} C_VEL
LIN {X 0,Y 453.552,Z 695.992,A -85,B 0,C 180,E1 -8296.196,E2 -8296.196} C_VEL
LIN {X 0,Y 453.524,Z 695.991,A -85,B 0,C 180,E1 -8299.039,E2 -8299.039} C_VEL
LIN {X 0,Y 453.484,Z 695.995,A -85,B 0,C 180,E1 -8301.836,E2 -8301.836} C_VEL
LIN {X 0,Y 453.508,Z 695.996,A -85,B 0,C 180,E1 -8304.735,E2 -8304.735} C_VEL
LIN {X 0,Y 453.513,Z 695.991,A -85,B 0,C 180,E1 -8307.953,E2 -8307.953} C_VEL
LIN {X 0,Y 453.482,Z 695.999,A -85,B 0,C 180,E1 -8310.759,E2 -8310.759} C_VEL
LIN {X 0,Y 453.475,Z 695.995,A -85,B 0,C 180,E1 -8313.913,E2 -8313.913} C_VEL
LIN {X 0,Y 453.459,Z 696.002,A -85,B 0,C 180,E1 -8317.189,E2 -8317.189} C_VEL
LIN {X 0,Y 453.512,Z 695.995,A -85,B 0,C 180,E1 -8319.448,E2 -8319.448} C_VEL
LIN {X 0,Y 453.469,Z 696,A -85,B 0,C 180,E1 -8322.994,E2 -8322.994} C_VEL
LIN {X 0,Y 453.468,Z 695.999,A -85,B 0,C 180,E1 -8325.778,E2 -8325.778} C_VEL
LIN {X 0,Y 453.485,Z 695.994,A -85,B 0,C 180,E1 -8328.209,E2 -8328.209} C_VEL
LIN {X 0,Y 453.476,Z 695.995,A -85,B 0,C 180,E1 -8330.796,E2 -8330.796} C_VEL
LIN {X 0,Y 453.457,Z 696.001,A -85,B 0,C 180,E1 -8333.916,E2 -8333.916} C_VEL
LIN {X 0,Y 453.484,Z 695.997,A -85,B 0,C 180,E1 -8337.15,E2 -8337.15} C_VEL
LIN {X 0,Y 453.535,Z 696.186,A -85,B 0,C 180,E1 -8338.783,E2 -8338.783} C_VEL
LIN {X 0,Y 457.04,Z 711.45,A -85,B 0,C 180,E1 -8341.223,E2 -8341.223} C_VEL
LIN {X 0,Y 458.089,Z 717.209,A -85,B 0,C 180,E1 -8342.099,E2 -8342.099} C_VEL
LIN {X 0,Y 456.906,Z 739.271,A -85,B 0,C 180,E1 -8345.165,E2 -8345.165} C_VEL
LIN {X 0,Y 455.916,Z 760.724,A -85,B 0,C 180,E1 -8348.104,E2 -8348.104} C_VEL
LIN {X 0,Y 454.801,Z 787.816,A -85,B 0,C 180,E1 -8351.763,E2 -8351.763} C_VEL
LIN {X 0,Y 454.629,Z 792.914,A -85,B 0,C 180,E1 -8352.419,E2 -8352.419} C_VEL
LIN {X 0,Y 457.453,Z 819.705,A -85,B 0,C 180,E1 -8352.969,E2 -8352.969} C_VEL
LIN {X 0,Y 456.74,Z 903.633,A -85,B 0,C 180,E1 -8354.32,E2 -8354.32} C_VEL
LIN {X 0,Y 456.211,Z 917.588,A -85,B 0,C 180,E1 -8354.731,E2 -8354.731} C_VEL
LIN {X 0,Y 455.753,Z 929.577,A -85,B 0,C 180,E1 -8355.258,E2 -8355.258} C_VEL
LIN {X 0,Y 455.129,Z 940.936,A -85,B 0,C 180,E1 -8355.923,E2 -8355.923} C_VEL
LIN {X 0,Y 454.63,Z 952.225,A -85,B 0,C 180,E1 -8356.775,E2 -8356.775} C_VEL
LIN {X 0,Y 454.139,Z 963.37,A -85,B 0,C 180,E1 -8357.826,E2 -8357.826} C_VEL
LIN {X 0,Y 453.655,Z 972.075,A -85,B 0,C 180,E1 -8358.833,E2 -8358.833} C_VEL
LIN {X 0,Y 453.278,Z 980.128,A -85,B 0,C 180,E1 -8359.953,E2 -8359.953} C_VEL
LIN {X 0,Y 453.031,Z 988.029,A -85,B 0,C 180,E1 -8361.299,E2 -8361.299} C_VEL
LIN {X 0,Y 452.86,Z 995.312,A -85,B 0,C 180,E1 -8362.867,E2 -8362.867} C_VEL
LIN {X 0,Y 452.811,Z 1000.172,A -85,B 0,C 180,E1 -8364.209,E2 -8364.209} C_VEL
LIN {X 0,Y 452.79,Z 1003.887,A -85,B 0,C 180,E1 -8365.548,E2 -8365.548} C_VEL
LIN {X 0,Y 452.814,Z 1005.807,A -85,B 0,C 180,E1 -8366.439,E2 -8366.439} C_VEL
LIN {X 0,Y 452.778,Z 1007.239,A -85,B 0,C 180,E1 -8367.33,E2 -8367.33} C_VEL
LIN {X 0,Y 452.775,Z 1008.257,A -85,B 0,C 180,E1 -8368.22,E2 -8368.22} C_VEL
LIN {X 0,Y 452.762,Z 1008.872,A -85,B 0,C 180,E1 -8369.109,E2 -8369.109} C_VEL
LIN {X 0,Y 452.766,Z 1009.084,A -85,B 0,C 180,E1 -8369.999,E2 -8369.999} C_VEL
LIN {X 0,Y 452.765,Z 1008.849,A -85,B 0,C 180,E1 -8370.888,E2 -8370.888} C_VEL
LIN {X 0,Y 452.781,Z 1008.209,A -85,B 0,C 180,E1 -8371.778,E2 -8371.778} C_VEL
LIN {X 0,Y 452.785,Z 1007.165,A -85,B 0,C 180,E1 -8372.668,E2 -8372.668} C_VEL
LIN {X 0,Y 452.813,Z 1005.71,A -85,B 0,C 180,E1 -8373.558,E2 -8373.558} C_VEL
LIN {X 0,Y 452.811,Z 1002.651,A -85,B 0,C 180,E1 -8374.896,E2 -8374.896} C_VEL
LIN {X 0,Y 452.819,Z 998.52,A -85,B 0,C 180,E1 -8376.236,E2 -8376.236} C_VEL
LIN {X 0,Y 452.907,Z 992.188,A -85,B 0,C 180,E1 -8377.802,E2 -8377.802} C_VEL
LIN {X 0,Y 453.099,Z 985.298,A -85,B 0,C 180,E1 -8379.147,E2 -8379.147} C_VEL
LIN {X 0,Y 453.399,Z 976.777,A -85,B 0,C 180,E1 -8380.493,E2 -8380.493} C_VEL
LIN {X 0,Y 453.729,Z 968.058,A -85,B 0,C 180,E1 -8381.615,E2 -8381.615} C_VEL
LIN {X 0,Y 454.356,Z 957.892,A -85,B 0,C 180,E1 -8382.681,E2 -8382.681} C_VEL
LIN {X 0,Y 454.868,Z 946.775,A -85,B 0,C 180,E1 -8383.627,E2 -8383.627} C_VEL
LIN {X 0,Y 455.416,Z 935.205,A -85,B 0,C 180,E1 -8384.408,E2 -8384.408} C_VEL
LIN {X 0,Y 455.963,Z 923.329,A -85,B 0,C 180,E1 -8385.018,E2 -8385.018} C_VEL
LIN {X 0,Y 456.474,Z 910.614,A -85,B 0,C 180,E1 -8385.486,E2 -8385.486} C_VEL
LIN {X 0,Y 456.784,Z 897.666,A -85,B 0,C 180,E1 -8385.79,E2 -8385.79} C_VEL
LIN {X 0,Y 457.325,Z 816.986,A -85,B 0,C 180,E1 -8387.072,E2 -8387.072} C_VEL
LIN {X 0,Y 454.6,Z 791.831,A -85,B 0,C 180,E1 -8387.608,E2 -8387.608} C_VEL
LIN {X 0,Y 455.456,Z 767.973,A -85,B 0,C 180,E1 -8390.786,E2 -8390.786} C_VEL
LIN {X 0,Y 456.368,Z 747.269,A -85,B 0,C 180,E1 -8393.601,E2 -8393.601} C_VEL
LIN {X 0,Y 457.461,Z 724.516,A -85,B 0,C 180,E1 -8396.746,E2 -8396.746} C_VEL
LIN {X 0,Y 457.919,Z 716.206,A -85,B 0,C 180,E1 -8397.91,E2 -8397.91} C_VEL
LIN {X 0,Y 454.647,Z 700.86,A -85,B 0,C 180,E1 -8400.312,E2 -8400.312} C_VEL
LIN {X 0,Y 453.508,Z 696.113,A -85,B 0,C 180,E1 -8401.124,E2 -8401.124} C_VEL
LIN {X 0,Y 453.471,Z 695.992,A -85,B 0,C 180,E1 -8403.911,E2 -8403.911} C_VEL
LIN {X 0,Y 453.446,Z 696.001,A -85,B 0,C 180,E1 -8407.188,E2 -8407.188} C_VEL
LIN {X 0,Y 453.482,Z 695.995,A -85,B 0,C 180,E1 -8409.448,E2 -8409.448} C_VEL
LIN {X 0,Y 453.469,Z 695.997,A -85,B 0,C 180,E1 -8411.934,E2 -8411.934} C_VEL
LIN {X 0,Y 453.485,Z 695.992,A -85,B 0,C 180,E1 -8415.469,E2 -8415.469} C_VEL
LIN {X 0,Y 453.473,Z 695.997,A -85,B 0,C 180,E1 -8418.208,E2 -8418.208} C_VEL
LIN {X 0,Y 453.501,Z 695.99,A -85,B 0,C 180,E1 -8420.79,E2 -8420.79} C_VEL
LIN {X 0,Y 453.447,Z 695.992,A -85,B 0,C 180,E1 -8423.916,E2 -8423.916} C_VEL
LIN {X 0,Y 453.473,Z 696.002,A -85,B 0,C 180,E1 -8427.15,E2 -8427.15} C_VEL
LIN {X 0,Y 453.503,Z 695.991,A -85,B 0,C 180,E1 -8430.27,E2 -8430.27} C_VEL
LIN {X 0,Y 453.519,Z 695.995,A -85,B 0,C 180,E1 -8433.295,E2 -8433.295} C_VEL
LIN {X 0,Y 453.492,Z 695.992,A -85,B 0,C 180,E1 -8436.238,E2 -8436.238} C_VEL
LIN {X 0,Y 453.471,Z 695.993,A -85,B 0,C 180,E1 -8439.117,E2 -8439.117} C_VEL
LIN {X 0,Y 453.5,Z 695.992,A -85,B 0,C 180,E1 -8441.944,E2 -8441.944} C_VEL
LIN {X 0,Y 453.537,Z 695.986,A -85,B 0,C 180,E1 -8444.726,E2 -8444.726} C_VEL
LIN {X 0,Y 453.548,Z 695.988,A -85,B 0,C 180,E1 -8448.379,E2 -8448.379} C_VEL
LIN {X 0,Y 453.639,Z 695.975,A -85,B 0,C 180,E1 -8451.985,E2 -8451.985} C_VEL
LIN {X 0,Y 453.656,Z 695.97,A -85,B 0,C 180,E1 -8454.667,E2 -8454.667} C_VEL
LIN {X 0,Y 453.754,Z 695.958,A -85,B 0,C 180,E1 -8457.337,E2 -8457.337} C_VEL
LIN {X 0,Y 453.81,Z 695.954,A -85,B 0,C 180,E1 -8460,E2 -8460} C_VEL
LIN {X 0,Y 453.753,Z 695.964,A -85,B 0,C 180,E1 -8462.663,E2 -8462.663} C_VEL
LIN {X 0,Y 453.657,Z 695.974,A -85,B 0,C 180,E1 -8466.226,E2 -8466.226} C_VEL
LIN {X 0,Y 453.581,Z 695.984,A -85,B 0,C 180,E1 -8468.914,E2 -8468.914} C_VEL
LIN {X 0,Y 453.551,Z 695.987,A -85,B 0,C 180,E1 -8472.529,E2 -8472.529} C_VEL
LIN {X 0,Y 453.532,Z 695.984,A -85,B 0,C 180,E1 -8476.197,E2 -8476.197} C_VEL
LIN {X 0,Y 453.506,Z 695.994,A -85,B 0,C 180,E1 -8479.04,E2 -8479.04} C_VEL
LIN {X 0,Y 453.465,Z 695.994,A -85,B 0,C 180,E1 -8481.837,E2 -8481.837} C_VEL
LIN {X 0,Y 453.484,Z 695.989,A -85,B 0,C 180,E1 -8484.736,E2 -8484.736} C_VEL
LIN {X 0,Y 453.518,Z 695.984,A -85,B 0,C 180,E1 -8487.96,E2 -8487.96} C_VEL
LIN {X 0,Y 453.457,Z 696.001,A -85,B 0,C 180,E1 -8491.526,E2 -8491.526} C_VEL
LIN {X 0,Y 453.48,Z 695.995,A -85,B 0,C 180,E1 -8494.779,E2 -8494.779} C_VEL
LIN {X 0,Y 453.465,Z 695.995,A -85,B 0,C 180,E1 -8498.312,E2 -8498.312} C_VEL
LIN {X 0,Y 453.486,Z 695.994,A -85,B 0,C 180,E1 -8500.61,E2 -8500.61} C_VEL
LIN {X 0,Y 453.447,Z 695.999,A -85,B 0,C 180,E1 -8503.245,E2 -8503.245} C_VEL
LIN {X 0,Y 453.453,Z 696.001,A -85,B 0,C 180,E1 -8505.78,E2 -8505.78} C_VEL
LIN {X 0,Y 453.509,Z 696.202,A -85,B 0,C 180,E1 -8507.734,E2 -8507.734} C_VEL
LIN {X 0,Y 453.772,Z 697.313,A -85,B 0,C 180,E1 -8507.881,E2 -8507.881} C_VEL
LIN {X 0,Y 457.999,Z 708.512,A -85,B 0,C 180,E1 -8508.254,E2 -8508.254} C_VEL
LIN {X 0,Y 457.44,Z 777.556,A -85,B 0,C 180,E1 -8509.382,E2 -8509.382} C_VEL
LIN {X 0,Y 457.328,Z 790.8,A -85,B 0,C 180,E1 -8509.786,E2 -8509.786} C_VEL
LIN {X 0,Y 457.144,Z 803.308,A -85,B 0,C 180,E1 -8510.352,E2 -8510.352} C_VEL
LIN {X 0,Y 456.86,Z 814.368,A -85,B 0,C 180,E1 -8511.024,E2 -8511.024} C_VEL
LIN {X 0,Y 456.409,Z 825.02,A -85,B 0,C 180,E1 -8511.849,E2 -8511.849} C_VEL
LIN {X 0,Y 455.963,Z 835.924,A -85,B 0,C 180,E1 -8512.913,E2 -8512.913} C_VEL
LIN {X 0,Y 455.366,Z 845.652,A -85,B 0,C 180,E1 -8514.094,E2 -8514.094} C_VEL
LIN {X 0,Y 454.856,Z 854.247,A -85,B 0,C 180,E1 -8515.403,E2 -8515.403} C_VEL
LIN {X 0,Y 454.487,Z 860.726,A -85,B 0,C 180,E1 -8516.62,E2 -8516.62} C_VEL
LIN {X 0,Y 454.166,Z 865.615,A -85,B 0,C 180,E1 -8517.734,E2 -8517.734} C_VEL
LIN {X 0,Y 453.797,Z 870.944,A -85,B 0,C 180,E1 -8519.266,E2 -8519.266} C_VEL
LIN {X 0,Y 453.623,Z 874.828,A -85,B 0,C 180,E1 -8520.791,E2 -8520.791} C_VEL
LIN {X 0,Y 453.454,Z 877.399,A -85,B 0,C 180,E1 -8522.294,E2 -8522.294} C_VEL
LIN {X 0,Y 453.338,Z 878.939,A -85,B 0,C 180,E1 -8524.049,E2 -8524.049} C_VEL
LIN {X 0,Y 453.314,Z 879.133,A -85,B 0,C 180,E1 -8525.256,E2 -8525.256} C_VEL
LIN {X 0,Y 453.289,Z 878.768,A -85,B 0,C 180,E1 -8526.229,E2 -8526.229} C_VEL
LIN {X 0,Y 453.317,Z 877.981,A -85,B 0,C 180,E1 -8527.177,E2 -8527.177} C_VEL
LIN {X 0,Y 452.731,Z 877.273,A -85,B 0,C 180,E1 -8527.916,E2 -8527.916} C_VEL
LIN {X 0,Y 450.022,Z 875.636,A -85,B 0,C 180,E1 -8529.11,E2 -8529.11} C_VEL
LIN {X 0,Y 447.756,Z 873.758,A -85,B 0,C 180,E1 -8530.057,E2 -8530.057} C_VEL
LIN {X 0,Y 446.85,Z 871.94,A -85,B 0,C 180,E1 -8530.77,E2 -8530.77} C_VEL
LIN {X 0,Y 446.814,Z 871.213,A -85,B 0,C 180,E1 -8531.008,E2 -8531.008} C_VEL
LIN {X 0,Y 447.186,Z 865.437,A -85,B 0,C 180,E1 -8532.628,E2 -8532.628} C_VEL
LIN {X 0,Y 447.555,Z 858.853,A -85,B 0,C 180,E1 -8534.051,E2 -8534.051} C_VEL
LIN {X 0,Y 448.074,Z 850.572,A -85,B 0,C 180,E1 -8535.467,E2 -8535.467} C_VEL
LIN {X 0,Y 448.541,Z 842.112,A -85,B 0,C 180,E1 -8536.641,E2 -8536.641} C_VEL
LIN {X 0,Y 449.043,Z 832.868,A -85,B 0,C 180,E1 -8537.689,E2 -8537.689} C_VEL
LIN {X 0,Y 449.48,Z 822.796,A -85,B 0,C 180,E1 -8538.616,E2 -8538.616} C_VEL
LIN {X 0,Y 449.972,Z 810.706,A -85,B 0,C 180,E1 -8539.496,E2 -8539.496} C_VEL
LIN {X 0,Y 450.287,Z 798.556,A -85,B 0,C 180,E1 -8540.172,E2 -8540.172} C_VEL
LIN {X 0,Y 450.443,Z 785.576,A -85,B 0,C 180,E1 -8540.686,E2 -8540.686} C_VEL
LIN {X 0,Y 450.52,Z 771.772,A -85,B 0,C 180,E1 -8541.027,E2 -8541.027} C_VEL
LIN {X 0,Y 450.996,Z 709.464,A -85,B 0,C 180,E1 -8542.038,E2 -8542.038} C_VEL
LIN {X 0,Y 446.729,Z 697.744,A -85,B 0,C 180,E1 -8542.43,E2 -8542.43} C_VEL
LIN {X 0,Y 446.571,Z 696.945,A -85,B 0,C 180,E1 -8542.598,E2 -8542.598} C_VEL
LIN {X 0,Y 446.624,Z 696.853,A -85,B 0,C 180,E1 -8544.584,E2 -8544.584} C_VEL
LIN {X 0,Y 446.66,Z 696.848,A -85,B 0,C 180,E1 -8548.198,E2 -8548.198} C_VEL
LIN {X 0,Y 446.721,Z 696.84,A -85,B 0,C 180,E1 -8550.001,E2 -8550.001} C_VEL
LIN {X 0,Y 446.653,Z 696.85,A -85,B 0,C 180,E1 -8552.707,E2 -8552.707} C_VEL
LIN {X 0,Y 446.609,Z 696.856,A -85,B 0,C 180,E1 -8556.326,E2 -8556.326} C_VEL
LIN {X 0,Y 446.51,Z 696.864,A -85,B 0,C 180,E1 -8559.057,E2 -8559.057} C_VEL
LIN {X 0,Y 446.527,Z 696.866,A -85,B 0,C 180,E1 -8562.731,E2 -8562.731} C_VEL
LIN {X 0,Y 446.489,Z 696.866,A -85,B 0,C 180,E1 -8566.46,E2 -8566.46} C_VEL
LIN {X 0,Y 446.439,Z 696.865,A -85,B 0,C 180,E1 -8569.306,E2 -8569.306} C_VEL
LIN {X 0,Y 446.421,Z 696.872,A -85,B 0,C 180,E1 -8572.201,E2 -8572.201} C_VEL
LIN {X 0,Y 446.414,Z 696.871,A -85,B 0,C 180,E1 -8575.156,E2 -8575.156} C_VEL
LIN {X 0,Y 446.421,Z 696.868,A -85,B 0,C 180,E1 -8578.184,E2 -8578.184} C_VEL
LIN {X 0,Y 446.394,Z 696.88,A -85,B 0,C 180,E1 -8581.303,E2 -8581.303} C_VEL
LIN {X 0,Y 446.417,Z 696.86,A -85,B 0,C 180,E1 -8584.525,E2 -8584.525} C_VEL
LIN {X 0,Y 446.392,Z 696.877,A -85,B 0,C 180,E1 -8587.882,E2 -8587.882} C_VEL
LIN {X 0,Y 446.401,Z 696.882,A -85,B 0,C 180,E1 -8591.396,E2 -8591.396} C_VEL
LIN {X 0,Y 446.422,Z 696.875,A -85,B 0,C 180,E1 -8595.109,E2 -8595.109} C_VEL
LIN {X 0,Y 446.402,Z 696.875,A -85,B 0,C 180,E1 -8598.605,E2 -8598.605} C_VEL
LIN {X 0,Y 446.39,Z 696.882,A -85,B 0,C 180,E1 -8602.119,E2 -8602.119} C_VEL
LIN {X 0,Y 446.389,Z 696.881,A -85,B 0,C 180,E1 -8605.473,E2 -8605.473} C_VEL
LIN {X 0,Y 446.395,Z 696.882,A -85,B 0,C 180,E1 -8608.698,E2 -8608.698} C_VEL
LIN {X 0,Y 446.451,Z 697.078,A -85,B 0,C 180,E1 -8609.752,E2 -8609.752} C_VEL
LIN {X 0,Y 446.666,Z 698.109,A -85,B 0,C 180,E1 -8609.894,E2 -8609.894} C_VEL
LIN {X 0,Y 450.505,Z 708.887,A -85,B 0,C 180,E1 -8610.242,E2 -8610.242} C_VEL
LIN {X 0,Y 449.89,Z 772.422,A -85,B 0,C 180,E1 -8611.354,E2 -8611.354} C_VEL
LIN {X 0,Y 449.74,Z 784.087,A -85,B 0,C 180,E1 -8611.694,E2 -8611.694} C_VEL
LIN {X 0,Y 449.464,Z 795.081,A -85,B 0,C 180,E1 -8612.151,E2 -8612.151} C_VEL
LIN {X 0,Y 449.296,Z 804.258,A -85,B 0,C 180,E1 -8612.645,E2 -8612.645} C_VEL
LIN {X 0,Y 448.911,Z 814.397,A -85,B 0,C 180,E1 -8613.326,E2 -8613.326} C_VEL
LIN {X 0,Y 448.545,Z 823.774,A -85,B 0,C 180,E1 -8614.103,E2 -8614.103} C_VEL
LIN {X 0,Y 448.091,Z 832.281,A -85,B 0,C 180,E1 -8614.945,E2 -8614.945} C_VEL
LIN {X 0,Y 447.741,Z 840.419,A -85,B 0,C 180,E1 -8615.913,E2 -8615.913} C_VEL
LIN {X 0,Y 447.43,Z 847.298,A -85,B 0,C 180,E1 -8616.878,E2 -8616.878} C_VEL
LIN {X 0,Y 447.042,Z 854.312,A -85,B 0,C 180,E1 -8618.058,E2 -8618.058} C_VEL
LIN {X 0,Y 446.718,Z 860.25,A -85,B 0,C 180,E1 -8619.269,E2 -8619.269} C_VEL
LIN {X 0,Y 446.579,Z 864.215,A -85,B 0,C 180,E1 -8620.223,E2 -8620.223} C_VEL
LIN {X 0,Y 446.339,Z 868.92,A -85,B 0,C 180,E1 -8621.644,E2 -8621.644} C_VEL
LIN {X 0,Y 446.206,Z 871.334,A -85,B 0,C 180,E1 -8622.587,E2 -8622.587} C_VEL
LIN {X 0,Y 446.08,Z 874.833,A -85,B 0,C 180,E1 -8624.464,E2 -8624.464} C_VEL
LIN {X 0,Y 446.037,Z 876.557,A -85,B 0,C 180,E1 -8626.329,E2 -8626.329} C_VEL
LIN {X 0,Y 446.075,Z 876.704,A -85,B 0,C 180,E1 -8627.644,E2 -8627.644} C_VEL
LIN {X 0,Y 446.13,Z 875.786,A -85,B 0,C 180,E1 -8629.103,E2 -8629.103} C_VEL
LIN {X 0,Y 446.226,Z 874.781,A -85,B 0,C 180,E1 -8630.023,E2 -8630.023} C_VEL
LIN {X 0,Y 446.289,Z 873.277,A -85,B 0,C 180,E1 -8630.939,E2 -8630.939} C_VEL
LIN {X 0,Y 446.581,Z 868.936,A -85,B 0,C 180,E1 -8632.767,E2 -8632.767} C_VEL
LIN {X 0,Y 446.802,Z 864.391,A -85,B 0,C 180,E1 -8634.132,E2 -8634.132} C_VEL
LIN {X 0,Y 447.037,Z 859.703,A -85,B 0,C 180,E1 -8635.265,E2 -8635.265} C_VEL
LIN {X 0,Y 447.346,Z 854.017,A -85,B 0,C 180,E1 -8636.397,E2 -8636.397} C_VEL
LIN {X 0,Y 447.777,Z 847.121,A -85,B 0,C 180,E1 -8637.526,E2 -8637.526} C_VEL
LIN {X 0,Y 448.18,Z 838.769,A -85,B 0,C 180,E1 -8638.652,E2 -8638.652} C_VEL
LIN {X 0,Y 448.591,Z 830.752,A -85,B 0,C 180,E1 -8639.551,E2 -8639.551} C_VEL
LIN {X 0,Y 449.026,Z 821.023,A -85,B 0,C 180,E1 -8640.448,E2 -8640.448} C_VEL
LIN {X 0,Y 449.367,Z 812.21,A -85,B 0,C 180,E1 -8641.12,E2 -8641.12} C_VEL
LIN {X 0,Y 449.661,Z 802.249,A -85,B 0,C 180,E1 -8641.735,E2 -8641.735} C_VEL
LIN {X 0,Y 449.951,Z 791.726,A -85,B 0,C 180,E1 -8642.238,E2 -8642.238} C_VEL
LIN {X 0,Y 450.033,Z 781.646,A -85,B 0,C 180,E1 -8642.601,E2 -8642.601} C_VEL
LIN {X 0,Y 450.094,Z 768.706,A -85,B 0,C 180,E1 -8642.909,E2 -8642.909} C_VEL
LIN {X 0,Y 450.885,Z 708.599,A -85,B 0,C 180,E1 -8643.978,E2 -8643.978} C_VEL
LIN {X 0,Y 446.672,Z 697.911,A -85,B 0,C 180,E1 -8644.397,E2 -8644.397} C_VEL
LIN {X 0,Y 446.508,Z 696.972,A -85,B 0,C 180,E1 -8644.57,E2 -8644.57} C_VEL
LIN {X 0,Y 446.625,Z 696.853,A -85,B 0,C 180,E1 -8646.324,E2 -8646.324} C_VEL
LIN {X 0,Y 446.527,Z 696.865,A -85,B 0,C 180,E1 -8649.97,E2 -8649.97} C_VEL
LIN {X 0,Y 446.529,Z 696.863,A -85,B 0,C 180,E1 -8652.729,E2 -8652.729} C_VEL
LIN {X 0,Y 446.503,Z 696.869,A -85,B 0,C 180,E1 -8656.227,E2 -8656.227} C_VEL
LIN {X 0,Y 446.476,Z 696.868,A -85,B 0,C 180,E1 -8659.303,E2 -8659.303} C_VEL
LIN {X 0,Y 446.425,Z 696.876,A -85,B 0,C 180,E1 -8662.199,E2 -8662.199} C_VEL
LIN {X 0,Y 446.45,Z 696.873,A -85,B 0,C 180,E1 -8665.153,E2 -8665.153} C_VEL
LIN {X 0,Y 446.456,Z 696.871,A -85,B 0,C 180,E1 -8668.181,E2 -8668.181} C_VEL
LIN {X 0,Y 446.422,Z 696.877,A -85,B 0,C 180,E1 -8671.3,E2 -8671.3} C_VEL
LIN {X 0,Y 446.429,Z 696.875,A -85,B 0,C 180,E1 -8674.523,E2 -8674.523} C_VEL
LIN {X 0,Y 446.422,Z 696.874,A -85,B 0,C 180,E1 -8678.079,E2 -8678.079} C_VEL
LIN {X 0,Y 446.434,Z 696.876,A -85,B 0,C 180,E1 -8680.917,E2 -8680.917} C_VEL
LIN {X 0,Y 446.407,Z 696.878,A -85,B 0,C 180,E1 -8683.845,E2 -8683.845} C_VEL
LIN {X 0,Y 446.402,Z 696.877,A -85,B 0,C 180,E1 -8686.403,E2 -8686.403} C_VEL
LIN {X 0,Y 446.433,Z 696.875,A -85,B 0,C 180,E1 -8689.082,E2 -8689.082} C_VEL
